# B&R Automation Studio project NAEUL004C00R13L518F00 (part 74)

#### InputRef.var - Do Not Change!!!
```iecst
(*2019-04-16*)
(**)
(*General*)
VAR
	p_udiRstErr : REFERENCE TO UDINT;
	p_bEn : REFERENCE TO BOOL;
	p_bDis : REFERENCE TO BOOL;
	p_bRun : REFERENCE TO BOOL;
	p_bStop : REFERENCE TO BOOL;
	p_bStep : REFERENCE TO BOOL;
END_VAR
(**)
(**)
VAR
	p_eUSCommMod1 : REFERENCE TO eMcSetCommMod;
	p_eUSCommMod2 : REFERENCE TO eMcSetCommMod;
	p_eUSCommMod3 : REFERENCE TO eMcSetCommMod;
	p_eDSCommMod1 : REFERENCE TO eMcSetCommMod;
	p_eDSCommMod2 : REFERENCE TO eMcSetCommMod;
	p_eDSCommMod3 : REFERENCE TO eMcSetCommMod;
END_VAR
(* *)
(**)
VAR
	p_tyBufferStat1 : REFERENCE TO tyBffrStat;
	p_tyBufferStat2 : REFERENCE TO tyBffrStat;
	p_tyBufferStat3 : REFERENCE TO tyBffrStat;
END_VAR
(**)
VAR
	p_dtBufferMagPresentTm1 : REFERENCE TO DATE_AND_TIME;
	p_dtBufferMagPresentTm2 : REFERENCE TO DATE_AND_TIME;
	p_dtBufferMagPresentTm3 : REFERENCE TO DATE_AND_TIME;
END_VAR
(* *)
VAR
	p_bUSHermesUSRdy1 : REFERENCE TO BOOL;
	p_bUSHermesUSGdRdy1 : REFERENCE TO BOOL;
	p_bUSHermesUSRdy2 : REFERENCE TO BOOL;
	p_bUSHermesUSGdRdy2 : REFERENCE TO BOOL;
	p_bUSHermesUSRdy3 : REFERENCE TO BOOL;
	p_bUSHermesUSGdRdy3 : REFERENCE TO BOOL;
	p_bUSSMEMAUSRdy1 : REFERENCE TO BOOL;
	p_bUSSMEMAUSRdy2 : REFERENCE TO BOOL;
	p_bUSSMEMAUSRdy3 : REFERENCE TO BOOL;
	p_bUSSMEMAGdBrdRdy1 : REFERENCE TO BOOL;
	p_bUSSMEMAGdBrdRdy2 : REFERENCE TO BOOL;
	p_bUSSMEMAGdBrdRdy3 : REFERENCE TO BOOL;
	p_bDSSMEMADSRdy1 : REFERENCE TO BOOL;
	p_bDSSMEMADSRdy2 : REFERENCE TO BOOL;
	p_bDSSMEMADSRdy3 : REFERENCE TO BOOL;
	p_bDSHermesDSRdy1 : REFERENCE TO BOOL;
	p_bDSHermesDSRdy2 : REFERENCE TO BOOL;
	p_bDSHermesDSRdy3 : REFERENCE TO BOOL;
	p_eULMod : REFERENCE TO eULMod;
	p_bBypsGdBadBrd : REFERENCE TO BOOL;
	p_bConvGdBrd : REFERENCE TO BOOL;
	p_usiLinkProdRcpCurrRcpMcMod : REFERENCE TO USINT;
	p_bOpsModGoneThrough : REFERENCE TO BOOL;
END_VAR
(**)
VAR
	p_tyParamTravLif : REFERENCE TO tyParamTravLifUL;
END_VAR
(**)
VAR
	p_sProgNm : REFERENCE TO STRING[15];
	p_bNtSettingsLoadDone : REFERENCE TO BOOL;
END_VAR
```

#### Local.var - Do Not Change!!!
```iecst
(*2019-04-16*)
(**)
(*Local Action, State & Status*)
VAR
	eStatus : eFBStatus := Idle;
	udiStatus : UDINT := 0;
END_VAR
(**)
(*Local Alarm*)
VAR
	tyAlmData : tyAlmDat;
	a_tyAlmText : ARRAY[10000..10099] OF tyAlmTxt;
END_VAR
(**)
(*Local Output*)
VAR
	sStepTxt : STRING[80];
	bPaused : BOOL;
END_VAR
(**)
(*Local Input*)
VAR
	udiRstErr : UDINT := 0;
	bEn : BOOL := TRUE;
	bDis : BOOL := FALSE;
	bRun : BOOL;
	bStop : BOOL;
	bStep : BOOL;
END_VAR
(*Insert your comment here.*)
VAR
	eUSCommMod1 : eMcSetCommMod;
	eUSCommMod2 : eMcSetCommMod;
	eUSCommMod3 : eMcSetCommMod;
	eDSCommMod1 : eMcSetCommMod;
	eDSCommMod2 : eMcSetCommMod;
	eDSCommMod3 : eMcSetCommMod;
	bUSSMEMAUSRdy3 : BOOL;
	bUSSMEMAGdBrdRdy3 : BOOL;
	udiUSPosAllwGo : UDINT := 99;
	udiDSPosAllwGo : UDINT := 99;
	a_bPosAllwSigOn : ARRAY[1..3] OF BOOL;
	a_udiPosAllwSum : ARRAY[1..3] OF UDINT;
	a_tyMagAllwBffrStat : ARRAY[1..3] OF tyBffrStat;
	a_udiMagAllwMagPresentTm : ARRAY[1..3] OF UDINT;
	a_udiMagAllwPriority : ARRAY[1..3] OF UDINT;
	udiMagPresentTm : UDINT;
	udiMagPresentTm1 : UDINT;
	bLocalUSRdy1 : BOOL;
	bLocalUSRdy2 : BOOL;
	bLocalUSRdy3 : BOOL;
	bLocalUSGdRdy1 : BOOL;
	bLocalUSGdRdy2 : BOOL;
	bLocalUSGdRdy3 : BOOL;
	bLocalDSRdy1 : BOOL;
	bLocalDSRdy2 : BOOL;
	bLocalDSRdy3 : BOOL;
	bDSHermesDSRdy1 : BOOL;
	bDSHermesDSRdy2 : BOOL;
	bDSHermesDSRdy3 : BOOL;
	bGdChk : BOOL;
	udi : UDINT;
END_VAR
(**)
(*Local*)
VAR
	sProgNm : STRING[80];
	bNtSettingsLoadDone : BOOL;
	bRstErr : BOOL;
	udiRstErrOld : UDINT;
	bInitDone : BOOL;
	bInitialDone : BOOL;
	eOpsStep : ePosUSAllwGoStep := ePosUSAllwGoStepNA;
	eGotoOpsStep : ePosUSAllwGoStep := ePosUSAllwGoUSCheck;
	eOpsStep1 : ePosDSAllwGoStep := ePosDSAllwGoStepNA;
	eGotoOpsStep1 : ePosDSAllwGoStep := ePosDSAllwGoDSCheck;
	fbMidChkDlyTm : TON := (PT:=T#1s);
	fbTopMidChkDlyTm : TON := (PT:=T#1s);
	udiCount : UDINT;
	udiCmpTm : UDINT;
	bBypsGdBadBrd : BOOL;
	eULMode : eULMod;
	bOpsModGonethrough : BOOL;
	udiModuleNum : UDINT;
END_VAR
```

### Simu.var - Change By Project
```iecst
(*2019-01-20*)
(**)
(*Action & State & Status*)
VAR
	p_SimuStat : UDINT;
	p_SimuStatus : UDINT;
	p_SimuStatTxt : UDINT;
END_VAR
(**)
(*Alarm*)
(**)
(*Output*)
VAR
	p_SimuSimuStatus : UDINT;
	p_SimuStatusRun : UDINT;
	p_SimuStatusStop : UDINT;
	p_SimuStatusCycleStop : UDINT;
	p_SimuStatusStep : UDINT;
	p_SimuRun : UDINT;
	p_SimuStop : UDINT;
	p_SimuStep : UDINT;
END_VAR
```

### Program Logical/Simulation/Simu (IEC, version 1.00.0) - 1.00.0 - 

#### Act_InitGlobal.st - Change By Project
```iecst
(** 2019-03-22 **)
ACTION Act_InitGlobal:

	(* Always Change If Project Change *)

	//Pass Data To Link
	p_eUISimuAct ACCESS p_UISimuAct;

	//Pass Data To Internal Use
	p_bLinkPaused ACCESS p_OpsPause;
	p_bNtSettingsLoadDone ACCESS p_StartupNtSettingsLoadDone;

	(* Always Change If Project Change *)

END_ACTION
```

#### InputRef_Link.var - Change By Project
```iecst
(*2019-01-20*)
(**)
VAR
	p_eUISimuAct : REFERENCE TO eSimulationsAction;
	p_bLinkPaused : REFERENCE TO BOOL;
END_VAR
```

#### Act_Link.st - Change By Project
```iecst
(** 2019-01-20 **)
ACTION Act_Link:

	p_bPaused := p_bLinkPaused;

END_ACTION
```

#### Local.var - Do Not Change!!!
```iecst
(*2019-04-30*)
(**)
(*Local Action, State & Status*)
VAR
	eAct : eSimulationsAction := SimulationsActIdle;
	eStat : eSimulationsAction := SimulationsActIdle;
	eStatus : eFBStatus := Idle;
	sStatTxt : STRING[200] := '';
	a_sStatText : ARRAY[0..50] OF STRING[200] := ['Idling','Starting Operations','Sequence Stopping Operations','Pause Operations In Step','Accepting New Data','Accepted New Data','Error Immediate Stop Operations',44('')];
END_VAR
(**)
(*Local Alarm*)
(**)
(*Local Output*)
VAR
	eSimuStatus : eSimulationsStatus := SimulationsStatusStop;
	bStatusRun : BOOL;
	bStatusStop : BOOL := TRUE;
	bStatusCycleStop : BOOL;
	bStatusStep : BOOL;
	bRun : BOOL;
	bStop : BOOL;
	bStep : BOOL;
END_VAR
(**)
(*Local Input*)
VAR
	udiRstErr : UDINT := 0;
	bPaused : BOOL;
	bNtSettingsLoadDone : BOOL := TRUE;
END_VAR
(**)
(*Local*)
VAR
	bRstErr : BOOL;
	udiRstErrOld : UDINT;
	bInitDone : BOOL;
	bInitialDone : BOOL;
	eStatOld : eSimulationsAction := SimulationsActIdle;
	usiStep : USINT;
END_VAR
```

### Simu1.var - Change By Project
```iecst
(*2022-10-17*)
(**)
(*Action & State & Status*)
(**)
(*Alarm*)
(**)
(*Output*)
VAR
	p_Simu1Paused : UDINT;
END_VAR
(**)
VAR
	p_Simu1InShutterAct : UDINT;
	p_Simu1OutShutterAct : UDINT;
	p_Simu1OutShutterAct2 : UDINT;
	p_Simu1OutShutterAct3 : UDINT;
END_VAR
```

### Simu1.typ - Do Not Change!!!
```iecst
(*2018-12-11*)
(**)
(*Sequence*)

TYPE
	eSimuRunStep :
		(
		SimuStepNA,
		SimuStepChkPshrRetSen,
		SimuStepChkSen,
		SimuStepInShutterRet,
		SimuStepInShutterExt,
		SimuStepOutShutterRet,
		SimuStepOutShutterExt
		);
END_TYPE
```

### Program Logical/Simulation/Simu1 (IEC) - 1.00.0 - 

#### InputRef.var
```iecst
(*2022-10-17*)
(**)
(*General*)
VAR
	p_udiRstErr : REFERENCE TO UDINT;
	p_bEn : REFERENCE TO BOOL;
	p_bDis : REFERENCE TO BOOL;
	p_bRun : REFERENCE TO BOOL;
	p_bStop : REFERENCE TO BOOL;
	p_bStep : REFERENCE TO BOOL;
END_VAR
(**)
(**)
VAR
	p_eInShuttStat : REFERENCE TO ePneuAction;
	p_eInShuttStatus : REFERENCE TO eFBStatus;
	p_eOutShuttStat : REFERENCE TO ePneuAction;
	p_eOutShuttStatus : REFERENCE TO eFBStatus;
	p_eOutShutt2Stat : REFERENCE TO ePneuAction;
	p_eOutShutt2Status : REFERENCE TO eFBStatus;
	p_eOutShutt3Stat : REFERENCE TO ePneuAction;
	p_eOutShutt3Status : REFERENCE TO eFBStatus;
END_VAR
(**)
(**)
VAR
	p_sProgNm : REFERENCE TO STRING[15];
	p_bNtSettingsLoadDone : REFERENCE TO BOOL;
END_VAR
```

#### Local.var
```iecst
(*2022-10-17*)
(**)
(*Local Action, State & Status*)
VAR
	eStatus : eFBStatus := Idle;
	udiStatus : UDINT := 0;
END_VAR
(**)
(*Local Alarm*)
VAR
	tyAlmData : tyAlmDat;
	a_tyAlmText : ARRAY[10000..10099] OF tyAlmTxt;
END_VAR
(**)
(*Local Output*)
VAR
	sStepTxt : STRING[80];
	bPaused : BOOL;
	ePshrAct : eMtrPshrAction;
	eInShutterAct : ePneuAction;
	eOutShutterAct : ePneuAction;
	eOutShutterAct2 : ePneuAction;
	eOutShutterAct3 : ePneuAction;
END_VAR
(**)
(*Local Input*)
VAR
	udiRstErr : UDINT := 0;
	bEn : BOOL := TRUE;
	bDis : BOOL := FALSE;
	bRun : BOOL;
	bStop : BOOL;
	bStep : BOOL;
END_VAR
(**)
(**)
VAR
	eInShutt1Stat : ePneuAction;
	eInShutt1Status : eFBStatus;
	eOutShutt2Stat : ePneuAction;
	eOutShutt2Status : eFBStatus;
	eOutShuttStat : ePneuAction;
	eOutShuttStatus : eFBStatus;
	eOutShutt3Stat : ePneuAction;
	eOutShutt3Status : eFBStatus;
END_VAR
(**)
VAR
	sProgNm : STRING[15];
	bNtSettingsLoadDone : BOOL := TRUE;
END_VAR
(**)
(*Local*)
VAR
	bRstErr : BOOL;
	udiRstErrOld : UDINT;
	bInitDone : BOOL;
	bInitialDone : BOOL;
	eSimuStep : eSimuRunStep := SimuStepNA;
	eSimuGotoStep : eSimuRunStep := SimuStepChkSen;
	fbShutterExtDlyTm : TON := (PT:=T#200ms);
	udiModuleNum : UDINT;
END_VAR
```

#### Act_InitGlobal.st
```iecst
(** 2022-10-17 **)
ACTION Act_InitGlobal:

	(* Always Change If Project Change *)

	//Pass Data To Link

	//Pass Data To Internal Use
	p_udiRstErr ACCESS p_RstErrReset;
	p_bRun ACCESS p_SimuRun;
	p_bStop ACCESS p_SimuStop;
	p_bStep ACCESS p_SimuStep;
	p_bNtSettingsLoadDone ACCESS p_StartupNtSettingsLoadDone;

	p_eInShuttStat ACCESS p_Pneu2SenInShutterStat;
	p_eInShuttStatus ACCESS p_Pneu2SenInShutterStatus;

	p_eOutShuttStat ACCESS p_Pneu2SenOutShutterStat;
	p_eOutShuttStatus ACCESS p_Pneu2SenOutShutterStatus;

	p_eOutShutt2Stat ACCESS p_Pneu2SenOutShutterStat2;
	p_eOutShutt2Status ACCESS p_Pneu2SenOutShutterStatus2;

	p_eOutShutt3Stat ACCESS p_Pneu2SenOutShutterStat3;
	p_eOutShutt3Status ACCESS p_Pneu2SenOutShutterStatus3;

	//p_sProgNm ACCESS p_NtParamSimuTeleNOProgNm;

	(* Always Change If Project Change *)

END_ACTION
```

#### Act_Initial.st
```iecst
(** 2022-10-17 **)
ACTION Act_Initial:

	//Initial

END_ACTION
```

#### Act_InitLocal.st
```iecst
(** 2022-10-17 **)
ACTION Act_InitLocal:

	//Input Reference Link To Local Variable
	p_udiRstErr ACCESS ADR(udiRstErr);
	p_bEn ACCESS ADR(bEn);
	p_bDis ACCESS ADR(bDis);
	p_bRun ACCESS ADR(bRun);
	p_bStop ACCESS ADR(bStop);
	p_bStep ACCESS ADR(bStep);

	p_eInShuttStat ACCESS ADR(eInShutt1Stat);
	p_eInShuttStatus ACCESS ADR(eInShutt1Status);
	p_eOutShuttStat ACCESS ADR(eOutShuttStat);
	p_eOutShuttStatus ACCESS ADR(eOutShuttStatus);
	p_eOutShutt2Stat ACCESS ADR(eOutShutt2Stat);
	p_eOutShutt2Status ACCESS ADR(eOutShutt2Status);
	p_eOutShutt3Stat ACCESS ADR(eOutShutt3Stat);
	p_eOutShutt3Status ACCESS ADR(eOutShutt3Status);

	p_sProgNm ACCESS ADR(sProgNm);
	p_bNtSettingsLoadDone ACCESS ADR(bNtSettingsLoadDone);

END_ACTION
```

#### Act_Link.st
```iecst
(** 2022-10-17 **)
ACTION Act_Link:

END_ACTION
```

#### Act_LinkEn.st
```iecst
(** 2022-10-17 **)
ACTION Act_LinkEn:

	//Link bPrep, bEn & bDis

END_ACTION
```

#### Cyclic.st
```iecst
(** 2022-10-17 **)
PROGRAM _CYCLIC

	IF bInitDone = FALSE THEN
		bInitDone	:= TRUE;

		Act_InitLocal;
		Act_InitGlobal;

	ELSIF bInitialDone = FALSE THEN
		IF p_bNtSettingsLoadDone = TRUE THEN
			bInitialDone	:= TRUE;

			Act_Initial;
		END_IF

	ELSE

		Act_RstErr;
		Act_LinkEn;
		Act_Link;
		Act_Background;
		Act_Alarm;

	END_IF

END_PROGRAM
```

#### Init.st
```iecst
(** 2022-10-17 **)
PROGRAM _INIT

	(* Always Change If Project Change *)

	//Pass Address To Global Address For External Use
	//Action, State & Status

	//Alarm

	//Output
	p_Simu1Paused					:= ADR(bPaused);

	p_Simu1InShutterAct				:= ADR(eInShutterAct);
	p_Simu1OutShutterAct			:= ADR(eOutShutterAct);
	p_Simu1OutShutterAct2			:= ADR(eOutShutterAct2);
	p_Simu1OutShutterAct3			:= ADR(eOutShutterAct2);

	(* Always Change If Project Change *)

END_PROGRAM
```

#### Program Logical/Simulation/Simu1/Sequence

##### Act_OpsInitial.st
```iecst
(** 2019-01-16 **)
ACTION Act_OpsInitial:

	eSimuGotoStep	:= SimuStepChkSen;
	eSimuStep		:= SimuStepNA;

END_ACTION
```

##### Act_OpsRst.st
```iecst
(** 2022-10-17 **)
ACTION Act_OpsRst:

	eOutShutterAct			:= PneuActIdle;
	eOutShutterAct2			:= PneuActIdle;
	eOutShutterAct3			:= PneuActIdle;
	fbShutterExtDlyTm(IN:=FALSE);

END_ACTION
```

##### Act_OpsRun.st
```iecst
(** 2022-10-17 **)
ACTION Act_OpsRun:

	IF eSimuGotoStep <> eSimuStep THEN

		CASE eSimuGotoStep OF

			ELSE
				eSimuStep	:= eSimuGotoStep;

		END_CASE

	END_IF

	IF eSimuGotoStep = eSimuStep THEN

		IF bPaused = FALSE THEN

			CASE eSimuStep OF

			SimuStepOutShutterExt:

						eOutShutterAct	:= PneuActExt;
						eOutShutterAct2 := PneuActExt;
						eOutShutterAct3	:= PneuActExt;

					IF 	p_eOutShuttStat = PneuActExt AND p_eOutShuttStatus = Done AND
						p_eOutShutt2Stat = PneuActExt AND p_eOutShutt2Status = Done AND
						p_eOutShutt3Stat = PneuActExt AND p_eOutShutt3Status = Done THEN

						eOutShutterAct	:= PneuActIdle;
						eOutShutterAct2 := PneuActIdle;
						eOutShutterAct3 := PneuActIdle;

						fbShutterExtDlyTm(IN:=TRUE);
						IF fbShutterExtDlyTm.Q THEN
							fbShutterExtDlyTm(IN:=FALSE);
						eSimuGotoStep	:= SimuStepOutShutterRet;
						END_IF
						bPaused				:= p_bStop OR p_bStep;
					END_IF

				SimuStepOutShutterRet:

					eOutShutterAct	:= PneuActRet;
					eOutShutterAct2 := PneuActRet;
					eOutShutterAct3 := PneuActRet;
					IF 	p_eOutShuttStat = PneuActRet AND p_eOutShuttStatus = Done AND
						p_eOutShutt2Stat = PneuActRet AND p_eOutShutt2Status = Done AND
						p_eOutShutt3Stat = PneuActRet AND p_eOutShutt3Status = Done	 THEN

						eOutShutterAct	:= PneuActIdle;
						eOutShutterAct2 := PneuActIdle;
						eOutShutterAct3 := PneuActIdle;

						fbShutterExtDlyTm(IN:=TRUE);
						IF fbShutterExtDlyTm.Q THEN
							fbShutterExtDlyTm(IN:=FALSE);
						eSimuGotoStep	:= SimuStepOutShutterExt;
						END_IF
						bPaused			:= p_bStop OR p_bStep;
					END_IF

			END_CASE

		END_IF
	END_IF

END_ACTION
```

### Simu2.var - Change By Project
```iecst
(*2022-10-17*)
(**)
(*Action & State & Status*)
(**)
(*Alarm*)
(**)
(*Output*)
VAR
	p_Simu2Paused : UDINT;
END_VAR
(**)
VAR
	p_Simu2DispCyclTmBffr1 : UDINT;
	p_Simu2DispCyclTmBffr2 : UDINT;
	p_Simu2DispCyclTmBffr3 : UDINT;
END_VAR
```

### Simu2.typ - Do Not Change!!!
```iecst
(*2018-12-11*)
(**)
(*Sequence*)
(*Display Buffer*)

TYPE
	tyDispBffrCycTm : 	STRUCT  (*Buffer Display in HMI*)
		diDispIdxSt : DINT; (*Start Index Display in HMI*)
		diDispIdxEnd : DINT; (*End Index Display in HMI*)
		a_tyDispBffrDat : ARRAY[1..c_diDispBffrSize]OF tyDispBffrCycTmDat; (*Array of Buffer Data Display in HMI*)
	END_STRUCT;
	tyDispBffrCycTmDat : 	STRUCT  (*Display Buffer Data*)
		sSlttoSltIdx : STRING[80]; (*Slot Index*)
		sCycleTm : STRING[80]; (*Board Loaded Time*)
		dwColor : DWORD; (*Color For Good & Bad Board*)
	END_STRUCT;
END_TYPE
```

### Program Logical/Simulation/Simu2 (IEC) - 1.00.0 - 

#### InputRef.var
```iecst
(*2022-10-17*)
(**)
(*General*)
VAR
	p_udiRstErr : REFERENCE TO UDINT;
	p_bEn : REFERENCE TO BOOL;
	p_bDis : REFERENCE TO BOOL;
	p_bRun : REFERENCE TO BOOL;
	p_bStop : REFERENCE TO BOOL;
	p_bStep : REFERENCE TO BOOL;
END_VAR
(**)
VAR
	p_diSltCap : REFERENCE TO DINT;
	p_diBffrTtlSlt : REFERENCE TO DINT;
	p_bTravDPosDiff : REFERENCE TO BOOL;
	p_bTravEPosDiff : REFERENCE TO BOOL;
	p_bTravFPosDiff : REFERENCE TO BOOL;
	p_bLifterBtmSltAPosDiff : REFERENCE TO BOOL;
	p_bLifterBtmSltBPosDiff : REFERENCE TO BOOL;
	p_bLifterBtmSltCPosDiff : REFERENCE TO BOOL;
	p_diLifterBtmCurrSltA : REFERENCE TO DINT;
	p_diLifterBtmCurrSltB : REFERENCE TO DINT;
	p_diLifterBtmCurrSltC : REFERENCE TO DINT;
	p_eOpsTravLifOpsStep : REFERENCE TO eTravLifULStep;
	p_eOpsTravLifGotoOpsStep : REFERENCE TO eTravLifULStep;
	p_dtTimeCurrDT : REFERENCE TO DATE_AND_TIME;
	p_uiTimeCurrDTStructMS : REFERENCE TO UINT;
	p_tyDispCycTmBffr : REFERENCE TO tyDispBffrCycTm;
	p_tyBuffer : REFERENCE TO tyBffr;
	p_diSlotCount : REFERENCE TO DINT;
END_VAR
(**)
(**)
(**)
VAR
	p_sProgNm : REFERENCE TO STRING[15];
	p_bNtSettingsLoadDone : REFERENCE TO BOOL;
END_VAR
```

#### Local.var
```iecst
(*2022-10-17*)
(**)
(*Local Action, State & Status*)
VAR
	eStatus : eFBStatus := Idle;
	udiStatus : UDINT := 0;
END_VAR
(**)
(*Local Alarm*)
VAR
	tyAlmData : tyAlmDat;
	a_tyAlmText : ARRAY[10000..10099] OF tyAlmTxt;
END_VAR
(**)
(*Local Output*)
VAR
	sStepTxt : STRING[80];
	bPaused : BOOL;
END_VAR
(**)
(*Local Input*)
VAR
	udiRstErr : UDINT := 0;
	bEn : BOOL := TRUE;
	bDis : BOOL := FALSE;
	bRun : BOOL;
	bStop : BOOL;
	bStep : BOOL;
END_VAR
(**)
VAR
	diSltCap : DINT := 1;
	diBffrTtlSlt : DINT;
	tyDispCycTmBffr : tyDispBffrCycTm;
	sCurrSlotTransition : STRING[80];
	diCnt : DINT;
	diSlotCount : DINT;
	diDispIdx : DINT;
	dicntr1 : DINT;
	a_tyDispCycTmBffr : ARRAY[0..2] OF tyDispBffrCycTm;
	tyBuffer : tyBffr;
	dtCycleTim : TIME;
	dtDumyTim : TIME := T#0ms;
	dwGdColor : DWORD;
	dwNAColor : DWORD;
	tAccumulateTimer : TIME;
	tPrevTim : TIME;
	sSltnumber : STRING[80];
	TtestPrevTim : DATE_AND_TIME;
	tTesttime : TIME;
	teststep : USINT;
	testpos : USINT;
END_VAR
(**)
(**)
VAR
	sProgNm : STRING[15];
	bNtSettingsLoadDone : BOOL := TRUE;
END_VAR
(**)
(*Local*)
VAR
	bRstErr : BOOL;
	udiRstErrOld : UDINT;
	bInitDone : BOOL;
	bInitialDone : BOOL;
	udiModuleNum : UDINT;
END_VAR
```

#### Act_Alarm.st
```iecst
(** 2022-10-17 **)
ACTION Act_Alarm:

	//Error
	IF EDGEPOS(eStatus = Error) THEN

		tyAlmData.sProgNm		:= p_sProgNm;
		tyAlmData.udiCode		:= udiStatus;
		tyAlmData.eSeverity		:= AlmSeverityError;
		tyAlmData.udiRunTime	:= tyAlmData.udiRunTime + 1;
		tyAlmData.bAlm			:= TRUE;
		tyAlmData.udiModuleNum  := udiModuleNum;
		g_sSimu1ProgNm		:= p_sProgNm;
		//Get Error Message
		IF tyAlmData.udiCode < 10000 OR tyAlmData.udiCode > 10099 THEN
			tyAlmData.sAlmMsg	:= 'Unknown';
			tyAlmData.sRcyMsg	:= 'Unknown';
		ELSE
			tyAlmData.sAlmMsg	:= a_tyAlmText[tyAlmData.udiCode].sAlmText;
			tyAlmData.sRcyMsg	:= a_tyAlmText[tyAlmData.udiCode].sRcyText;
		END_IF

	ELSIF bRstErr AND (tyAlmData.udiCode <> 0) THEN

		tyAlmData.udiCode		:= 0;
		tyAlmData.eSeverity		:= AlmSeverityNA;
		tyAlmData.sAlmMsg		:= '';
		tyAlmData.sRcyMsg		:= '';
		tyAlmData.bAlm			:= FALSE;
	END_IF

END_ACTION
```

#### Act_Background.st
```iecst
(** 2022-10-17 **)
ACTION Act_Background:

	//Reset bPaused
	IF EDGENEG(p_bStop OR p_bStep) THEN
		bPaused	:= FALSE;
	END_IF

	IF eStatus <> Error AND p_bRun = TRUE THEN
		IF (p_bEn = TRUE) AND (p_bDis = FALSE) THEN
			Act_OpsRun;
		ELSE
			bPaused	:= p_bStop OR p_bStep;
		END_IF

		IF EDGEPOS(p_bEn = FALSE OR p_bDis = TRUE) THEN
			Act_OpsRst;
		END_IF

	ELSIF eStatus <> Error THEN
		sStepTxt	:= 'Stop';
	ELSE
		sStepTxt	:= 'Error';
	END_IF

	//Reset
	IF EDGENEG(p_bRun) OR EDGEPOS(eStatus = Error) THEN
		Act_OpsInitial;
		Act_OpsRst;
	END_IF

	//Reset Error
	IF (eStatus = Error) AND bRstErr THEN
		eStatus		:= Idle;
		udiStatus	:= 0;
	END_IF

END_ACTION
```

#### Act_InitGlobal.st
```iecst
(** 2022-10-17 **)
ACTION Act_InitGlobal:

	(* Always Change If Project Change *)

	//Pass Data To Link

	//Pass Data To Internal Use
	p_udiRstErr ACCESS p_RstErrReset;
	p_bRun ACCESS p_SimuRun;
	p_bStop ACCESS p_SimuStop;
	p_bStep ACCESS p_SimuStep;
	p_bNtSettingsLoadDone ACCESS p_StartupNtSettingsLoadDone;

	//OpsCycleTim
	p_bTravDPosDiff ACCESS p_TravDPosDiff;
	p_bTravEPosDiff ACCESS p_TravEPosDiff;
	p_bTravFPosDiff ACCESS p_TravFPosDiff;
	p_bLifterBtmSltAPosDiff ACCESS p_LifterBtmSltAPosDiff;
	p_bLifterBtmSltBPosDiff ACCESS p_LifterBtmSltBPosDiff;
	p_bLifterBtmSltCPosDiff ACCESS p_LifterBtmSltCPosDiff;
	p_diLifterBtmCurrSltA ACCESS p_LifterBtmCurrSltA;
	p_diLifterBtmCurrSltB ACCESS p_LifterBtmCurrSltB;
	p_diLifterBtmCurrSltC ACCESS p_LifterBtmCurrSltC;

	p_eOpsTravLifOpsStep ACCESS p_OpsTravLifOpsStep;
	p_eOpsTravLifGotoOpsStep ACCESS p_OpsTravLifGotoOpsStep;
	p_dtTimeCurrDT ACCESS p_TimeCurrDT	;
	p_diBffrTtlSlt ACCESS p_MagRcpCurrRcpTtlSlt;
    p_uiTimeCurrDTStructMS ACCESS p_TimeCurrDTStructMS;
	//p_sProgNm ACCESS p_NtParamSimuTeleNOProgNm;

	(* Always Change If Project Change *)

END_ACTION
```

#### Act_InitLocal.st
```iecst
(** 2022-10-17 **)
ACTION Act_InitLocal:

	//Input Reference Link To Local Variable
	p_udiRstErr ACCESS ADR(udiRstErr);
	p_bEn ACCESS ADR(bEn);
	p_bDis ACCESS ADR(bDis);
	p_bRun ACCESS ADR(bRun);
	p_bStop ACCESS ADR(bStop);
	p_bStep ACCESS ADR(bStep);

	p_diSltCap ACCESS ADR(diSltCap);
	p_diBffrTtlSlt ACCESS ADR(diBffrTtlSlt);
	p_tyDispCycTmBffr ACCESS ADR(tyDispCycTmBffr);
	p_tyBuffer ACCESS ADR(tyBuffer);
	p_diSltCap ACCESS ADR(diSltCap);
	p_diSlotCount ACCESS ADR(diCnt);

	p_sProgNm ACCESS ADR(sProgNm);
	p_bNtSettingsLoadDone ACCESS ADR(bNtSettingsLoadDone);

END_ACTION
```

#### Act_Link.st
```iecst
(** 2022-10-17 **)
ACTION Act_Link:

 	//tTesttime := UINT_TO_TIME(p_uiTimeCurrDTStructMS);
END_ACTION
```

#### Act_RstErr.st
```iecst
(** 2022-10-17 **)
ACTION Act_RstErr:

	IF p_udiRstErr <> udiRstErrOld THEN
		bRstErr			:= TRUE;
		udiRstErrOld	:= p_udiRstErr;
	ELSE
		bRstErr			:= FALSE;
	END_IF

END_ACTION
```

#### Init.st
```iecst
(** 2022-10-17 **)
PROGRAM _INIT

	(* Always Change If Project Change *)

	//Pass Address To Global Address For External Use
	//Action, State & Status

	//Alarm

	//Output
	p_Simu2Paused					:= ADR(bPaused);

	p_Simu2DispCyclTmBffr1					:= ADR(a_tyDispCycTmBffr[0]);
	p_Simu2DispCyclTmBffr2					:= ADR(a_tyDispCycTmBffr[1]);
	p_Simu2DispCyclTmBffr3					:= ADR(a_tyDispCycTmBffr[2]);

	(* Always Change If Project Change *)

END_PROGRAM
```

#### Act_OpsInitial.st - Do Not Change!!!
```iecst
(** 2019-01-16 **)
ACTION Act_OpsInitial:

END_ACTION
```

#### Act_OpsRun.st
```iecst
(** 2022-10-17 **)
ACTION Act_OpsRun:

	//A15<-A13 | timetaken

	IF (p_eOpsTravLifOpsStep =  TravLifULStepExitBrd AND p_eOpsTravLifGotoOpsStep = TravLifULStepOutletPneuCls)  THEN
		memset(ADR(dtCycleTim),0,SIZEOF(dtCycleTim));
		IF FIND(sCurrSlotTransition,'<-') <> 0 THEN
			sCurrSlotTransition := LEFT( sCurrSlotTransition , FIND(sCurrSlotTransition,'<-') - 1);
		END_IF

		IF NOT(p_bTravDPosDiff  OR p_bLifterBtmSltAPosDiff)   THEN
			itoa(DINT_TO_INT(p_diLifterBtmCurrSltA),ADR(sSltnumber));
			sCurrSlotTransition := CONCAT(CONCAT(CONCAT('A',sSltnumber),'<-'),sCurrSlotTransition);
			dtCycleTim := ((DT_TO_TIME(p_dtTimeCurrDT) +UINT_TO_TIME(p_uiTimeCurrDTStructMS) -tPrevTim )+ tAccumulateTimer);
			tPrevTim 			:= DT_TO_TIME(p_dtTimeCurrDT) + UINT_TO_TIME(p_uiTimeCurrDTStructMS);
		ELSIF NOT(p_bTravEPosDiff OR p_bLifterBtmSltBPosDiff )  THEN
			itoa(DINT_TO_INT(p_diLifterBtmCurrSltB),ADR(sSltnumber));
			sCurrSlotTransition := CONCAT(CONCAT(CONCAT('B',sSltnumber),'<-'),sCurrSlotTransition);
			dtCycleTim := ((DT_TO_TIME(p_dtTimeCurrDT) +UINT_TO_TIME(p_uiTimeCurrDTStructMS) -tPrevTim )+ tAccumulateTimer);
			tPrevTim 			:= DT_TO_TIME(p_dtTimeCurrDT) + UINT_TO_TIME(p_uiTimeCurrDTStructMS);
		ELSIF NOT(p_bTravFPosDiff OR p_bLifterBtmSltCPosDiff)  THEN
			itoa(DINT_TO_INT(p_diLifterBtmCurrSltC),ADR(sSltnumber));
			sCurrSlotTransition := CONCAT(CONCAT(CONCAT('C',sSltnumber),'<-'),sCurrSlotTransition);
			dtCycleTim := ((DT_TO_TIME(p_dtTimeCurrDT) +UINT_TO_TIME(p_uiTimeCurrDTStructMS) -tPrevTim )+ tAccumulateTimer); //+ tAccumulateTimer
			tPrevTim 			:= DT_TO_TIME(p_dtTimeCurrDT) + UINT_TO_TIME(p_uiTimeCurrDTStructMS);
		ELSE
			sCurrSlotTransition := '';
			tPrevTim 			:= 0;
		END_IF
		IF memcmp(ADR(dtCycleTim),ADR(dtDumyTim),SIZEOF(dtCycleTim)) <> 0 THEN ;
			Act_DispBffr;
		END_IF
	ELSIF (p_eOpsTravLifGotoOpsStep = TravLifULStepUSComm AND (p_eOpsTravLifOpsStep = TravLifULStepInletPneuOpn OR p_eOpsTravLifOpsStep= TravLifULStepTravLifMov ))  THEN
			IF tPrevTim <> 0 THEN
				tAccumulateTimer := (DT_TO_TIME(p_dtTimeCurrDT)+UINT_TO_TIME(p_uiTimeCurrDTStructMS) ) - tPrevTim  ;
			END_IF
	ELSIF (p_eOpsTravLifOpsStep =  TravLifULStepUSComm AND p_eOpsTravLifGotoOpsStep = TravLifULStepEntBrd) THEN
			tPrevTim		  := DT_TO_TIME(p_dtTimeCurrDT) +UINT_TO_TIME(p_uiTimeCurrDTStructMS) ;
	END_IF

END_ACTION
```

#### Act_OpsRst.st - Do Not Change!!!
```iecst
(** 2022-10-17 **)
ACTION Act_OpsRst:

	tPrevTim := 0;
	tAccumulateTimer := 0;

END_ACTION
```

#### Act_DispBffr.st
```iecst
(** 2022-10-17 **)
ACTION Act_DispBffr:

	memset(ADR(p_tyDispCycTmBffr) , 0 , SIZEOF(p_tyDispCycTmBffr));
	IF NOT(p_bTravDPosDiff  OR p_bLifterBtmSltAPosDiff) THEN
		p_tyDispCycTmBffr ACCESS ADR(a_tyDispCycTmBffr[0]);
		p_tyBuffer ACCESS p_Buffer1Bffr;
		p_diSlotCount ACCESS p_LifterBtmCurrSltA;
	ELSIF NOT(p_bTravEPosDiff OR p_bLifterBtmSltBPosDiff ) THEN
		p_tyDispCycTmBffr ACCESS ADR(a_tyDispCycTmBffr[1]);
		p_tyBuffer ACCESS p_Buffer2Bffr;
		p_diSlotCount ACCESS p_LifterBtmCurrSltB;
	ELSIF NOT(p_bTravFPosDiff OR p_bLifterBtmSltCPosDiff) THEN
		p_tyDispCycTmBffr ACCESS ADR(a_tyDispCycTmBffr[2]);
		p_tyBuffer ACCESS p_Buffer3Bffr;
		p_diSlotCount ACCESS p_LifterBtmCurrSltC;
	END_IF
	diCnt	:= 0;
	dwNAColor := 0;
	dwGdColor := 1;

	FOR dicntr1 := 1 TO p_diBffrTtlSlt DO

		//Get Display Index
		diDispIdx	:= p_diBffrTtlSlt * p_diSltCap - diCnt; //p_diLifterBtmCurrSltA
		diCnt := diCnt +1;

		IF p_diSlotCount = diCnt AND p_tyBuffer.a_tyBffrDat[diCnt].bSltForBrd AND p_tyBuffer.a_tyBffrDat[diCnt].bBrdAvl AND p_tyBuffer.a_tyBffrDat[diCnt].a_tySubBffrDat[1].bSubForBrd AND p_tyBuffer.a_tyBffrDat[diCnt].a_tySubBffrDat[1].bBrdAvl THEN
			ascTIME(dtCycleTim , ADR(p_tyDispCycTmBffr.a_tyDispBffrDat[diDispIdx].sCycleTm) , SIZEOF(p_tyDispCycTmBffr.a_tyDispBffrDat[diDispIdx].sCycleTm));
			p_tyDispCycTmBffr.a_tyDispBffrDat[diDispIdx].dwColor	:= dwGdColor;
			p_tyDispCycTmBffr.a_tyDispBffrDat[diDispIdx].sSlttoSltIdx := sCurrSlotTransition;
		ELSE
			p_tyDispCycTmBffr.a_tyDispBffrDat[diDispIdx].dwColor	:= dwNAColor;
			p_tyDispCycTmBffr.a_tyDispBffrDat[diDispIdx].sSlttoSltIdx := DINT_TO_STRING(dicntr1);
		END_IF

	END_FOR

	p_tyDispCycTmBffr.diDispIdxSt	:= 1;
	p_tyDispCycTmBffr.diDispIdxEnd	:= p_diBffrTtlSlt * p_diSltCap;

END_ACTION
```

### OpCon.typ - Do Not Change!!!
```iecst
(*2019-05-04*)
(**)
(*Action*)

TYPE
	eOpConAction :
		(
		OpConActIdle,
		OpConActBGStartRun,
		OpConActBGStopRun,
		OpConActDeleteOldLog,
		OpConActCreateDir,
		OpConActWriteRetain,
		OpConActReadRetain,
		OpConActWriteConfig,
		OpConActReadConfig
		);
END_TYPE
```

### OpCon.var - Change By Project
```iecst
(*2019-06-10*)
(**)
(*Action & State & Status*)
VAR
	p_OpConStat : UDINT;
	p_OpConStatus : UDINT;
	p_OpConStatTxt : UDINT;
END_VAR
(**)
(*Alarm*)
VAR
	p_OpConAlmData : UDINT;
	p_OpConAlmData1 : UDINT;
	p_OpConInfoData : UDINT;
END_VAR
(**)
(*Output*)
VAR
	p_OpConTableDataBrdAvl : UDINT;
	p_OpConTableDataBrdAvlTtlIdx : UDINT;
	p_OpConConnected : UDINT;
	p_OpConHandshakeDone : UDINT;
	p_OpConOverWriteSlt : UDINT;
	p_OpConOverWriteWidth : UDINT;
	p_OpConReqRecipeNm : UDINT;
	p_OpConReqWidthInUM : UDINT;
	p_OpConInternalSnd : UDINT;
	p_OpConPartRcvRetCode : UDINT;
	p_OpConPlcGrabRcvCode : UDINT;
END_VAR
```

### Program Logical/OpCon/OpCon (IEC, version 1.00.0) - 1.00.0 - NtHermes v5.00.0 , NtTCP v5.00.0 , NtMessage v5.00.0

#### Init.st - Change By Project
```iecst
(** 2019-06-10 **)
PROGRAM _INIT

	(* Always Change If Project Change *)

	//Pass Address To Global Address For External Use
	//Action, State & Status
	p_OpConStat		:= ADR(eStat);
	p_OpConStatus	:= ADR(eMainStatus);
	p_OpConStatTxt	:= ADR(sStatTxt);

	//Alarm
	p_OpConAlmData	:= ADR(tyAlmData);
	p_OpConAlmData1	:= ADR(tyAlmData1);
	p_OpConInfoData	:= ADR(tyInfoData);

	//Output
	p_OpConTableDataBrdAvl			:= ADR(a_tyXMLTableDataBrdAvl);
	p_OpConTableDataBrdAvlTtlIdx	:= ADR(iXMLTableDataBrdAvlTtlIdx);
	p_OpConConnected				:= ADR(bConnected);
	p_OpConHandshakeDone			:= ADR(bHandshakeDone);
	p_OpConOverWriteSlt			:= ADR(bOverWriteSlt);
	p_OpConOverWriteWidth		:= ADR(bOverWriteWidth);
	p_OpConReqRecipeNm			:= ADR(sReqRecipeNm);
	p_OpConReqWidthInUM			:= ADR(diReqWidthInUM);
	p_OpConInternalSnd			:= ADR(sInternalSnd);

	p_OpConPartRcvRetCode		:= ADR(tyPartReceive);
	p_OpConPlcGrabRcvCode			:= ADR(tyPlcGrab);
	(* Always Change If Project Change *)

END_PROGRAM
```

#### Act_InitGlobal.st - Change By Project
```iecst
(** 2019-06-28 **)
ACTION Act_InitGlobal:

	(* Always Change If Project Change *)

	//Pass Data To Link
	p_bLinkStartupRun ACCESS p_StartupRun;

	p_eLinkConvDir ACCESS p_NtParamProjConvDir;
	p_bLinkDILeftSen ACCESS p_DIConvLftSen;
	p_bLinkDIRightSen ACCESS p_DIConvRgtSen;
	p_tyLinkAlarmCurrList ACCESS p_AlarmCurrList;
	p_bLinkOpConEn ACCESS p_McParamOpConEn;

	//Pass Data To Internal Use
	p_udiRstErr ACCESS p_RstErrReset;
	p_bPrep ACCESS p_NtParamProjOpConPrep;
//	p_bEn ACCESS p_McParamOpConEn;
	p_sIPAddr ACCESS p_HWInfoIPAddr; //client
	p_sSvrIPAddr ACCESS p_McParamOpConIP;
	p_uiSvrIPPort ACCESS p_McParamOpConPort;
	p_tyDTStructure ACCESS p_TimeCurrDTStruct;
	p_dtCurrDT ACCESS p_TimeCurrDT;

	p_sRecipeNm ACCESS p_ProdRcpCurrRcp0Nm;
	p_diWidthInUM ACCESS p_ProdRcpCurrRcp0Width;
	p_bOpsRun ACCESS p_OpsRun;
	p_bNtSettingsLoadDone ACCESS p_StartupNtSettingsLoadDone;
	pa_tyProdRcpList ACCESS p_ProdRcpCurrList;
	p_tyProdRcpCurrRcp ACCESS p_ProdRcpCurrRcp0;

	p_tyOpConLocation ACCESS p_McParamOpConParam;
	p_bOpsTravLifULExitBrd ACCESS p_OpsTravLifULExitBrd;
	p_tyOpsTravLifULMsgReq ACCESS p_OpsTravLifULMsgReq;
	p_sOpsTravLifULBarcode ACCESS p_OpsTravLifULBarcode;
	p_tyOpsTravLifULPartProcessItms ACCESS p_OpsTravLifULPartProcessItms; //new
	pas_OpsTravLifULMagEntered ACCESS p_OpsTravLifULMagEntered;
	p_tyOpsMagConvUL1MsgReq ACCESS p_OpsMagConvUL1MsgReq;
	(* Always Change If Project Change *)

END_ACTION
```

#### InputRef_Link.var - Change By Project
```iecst
(*2019-04-16*)
(**)
VAR
	p_bLinkStartupRun : REFERENCE TO BOOL;
	bOpConRun : BOOL;
	bOpConStop : BOOL;
END_VAR
(**)
VAR
	p_eLinkConvDir : REFERENCE TO eConvDir;
	p_bLinkDILeftSen : REFERENCE TO BOOL;
	p_bLinkDIRightSen : REFERENCE TO BOOL;
	sWidthInUMTemp : STRING[80];
END_VAR
(**)
VAR
	p_tyLinkAlarmCurrList : REFERENCE TO ARRAY[1..c_udiAlarmCurrMax] OF tyAlarmCurr;
	p_bLinkOpConEn : REFERENCE TO BOOL;
END_VAR
```

#### Act_LinkAction.st - Change By Project
```iecst
(** 2019-04-09 **)
ACTION Act_LinkAction:

	IF p_bLinkStartupRun = TRUE THEN
	//	p_eAct ACCESS p_StartupUSOpConAct;
	ELSE
		p_eAct ACCESS ADR(eAct);

		IF p_bLinkOpConEn THEN
			bOpConRun	:= TRUE;
			bOpConStop	:= FALSE;
		ELSE
			bOpConRun	:= FALSE;
			bOpConStop	:= TRUE;
		END_IF

//		IF EDGEPOS(p_eLinkMcParamUSCommMod = McSetCommModOpCon) THEN
//			bOpConRun	:= TRUE;
//			bOpConStop	:= FALSE;
//		END_IF
//
//		IF EDGENEG(p_eLinkMcParamUSCommMod = McSetCommModOpCon) THEN
//			bOpConRun	:= FALSE;
//			bOpConStop	:= TRUE;
//		END_IF

		IF bOpConRun = TRUE THEN
			p_eAct	:= OpConActBGStartRun;

			IF (eStat = OpConActBGStartRun) AND (eStatus = Done) THEN
				p_eAct		:= OpConActIdle;
				bOpConRun	:= FALSE;
			END_IF
		END_IF

		IF bOpConStop = TRUE THEN
			p_eAct	:= OpConActBGStopRun;

			IF (eStat = OpConActBGStopRun) AND (eStatus = Done) THEN
				p_eAct		:= OpConActIdle;
				bOpConStop	:= FALSE;
			END_IF
		END_IF

	END_IF

END_ACTION
```

#### Act_Link.st - Change By Project
```iecst
(** 2019-06-04 **)
ACTION Act_Link:
	IF tyPartReceive.tyData.sTypeNo <> '' AND tyPartReceive.tyData.sTypeVar <> '' THEN
		tyPartProcessed.tyData.sTypeNo 		:= tyPartReceive.tyData.sTypeNo;
		tyPartProcessed.tyData.sTypeVar 	:= tyPartReceive.tyData.sTypeVar;
		tyPLCError.tyData.sTypeNo  			:= tyPartReceive.tyData.sTypeNo;
		tyPLCError.tyData.sTypeVar  		:= tyPartReceive.tyData.sTypeVar;
		tyPartMissing.tyData.sTypeNo  		:= tyPartReceive.tyData.sTypeNo;
		tyPartMissing.tyData.sTypeVar  		:= tyPartReceive.tyData.sTypeVar;
		tyPLCJam.tyData.sTypeNo  			:= tyPartReceive.tyData.sTypeNo;
		tyPLCJam.tyData.sTypeVar  			:= tyPartReceive.tyData.sTypeVar;
	END_IF

	IF p_bOpsTravLifULExitBrd THEN
		tyPartReceive.tyAvl.bReturnCode				:= FALSE;
	END_IF

END_ACTION
```

#### Cyclic.st - Do Not Change!!!
```iecst
(** 2019-04-21 **)
PROGRAM _CYCLIC

	IF bInitDone = FALSE THEN
		bInitDone	:= TRUE;

		Act_InitLocal;
		Act_InitGlobal;

	ELSIF bInitialDone = FALSE THEN
		IF p_bNtSettingsLoadDone = TRUE THEN
			bInitialDone	:= TRUE;

			Act_Initial;
		END_IF

	ELSE

		Act_RstErr;
		Act_LinkAction;
		Act_Action;
		Act_LinkEn;

		IF (p_bPrep = TRUE) AND (p_bEn = TRUE) AND (p_bDis = FALSE) THEN
			Act_Link;
			Act_Main;
			Act_Background;

		ELSE
			Act_Main_Disable;

			IF eStat <> OpConActIdle THEN
				eStatus	:= Done;
			ELSE
				eStatus	:= Idle;
			END_IF
		END_IF

		Act_CombineErr;
		Act_Alarm;
		Act_Alarm1;
	END_IF

END_PROGRAM
```

#### Act_InitLocal.st - Do Not Change!!!
```iecst
(** 2019-06-28 **)
ACTION Act_InitLocal:

	//Input Reference Link To Local Variable
	p_eAct ACCESS ADR(eAct);
	p_udiRstErr ACCESS ADR(udiRstErr);
	p_bPrep ACCESS ADR(bPrep);
	p_bEn ACCESS ADR(bEn);
	p_bDis ACCESS ADR(bDis);
	p_sIPAddr ACCESS ADR(sIPAddr);
	p_uiClntPort ACCESS ADR(uiClntPort); //def :0
	p_tyDTStructure ACCESS ADR(tyDTStructure);
	p_dtCurrDT ACCESS ADR(dtCurrDT);
	p_sVersion ACCESS ADR(sVersion);
	p_sRecipeNm ACCESS ADR(sRecipeNm);
	p_diWidthInUM ACCESS ADR(diWidthInUM);
	p_udiSndBffrSize ACCESS ADR(udiSndBffrSize);
	p_udiRcvBffrSize ACCESS ADR(udiRcvBffrSize);
	p_udiAliveIdleTimeInSec ACCESS ADR(udiAliveIdleTimeInSec);
	p_tConnTimeOut ACCESS ADR(tConnTimeOut);
	p_diTransferInTO ACCESS ADR(diTransferInTO);
	p_bOpsRun ACCESS ADR(bOpsRun);
	p_bInterruptSen ACCESS ADR(bInterruptSen);
	p_udiFileKeepDay ACCESS ADR(udiFileKeepDay);
	p_sProgNm ACCESS ADR(sProgNm);
	p_bNtSettingsLoadDone ACCESS ADR(bNtSettingsLoadDone);
	p_sInfoMsg ACCESS ADR(sInfoMsg);
	p_bInternalUse ACCESS ADR(bInternalUse);
	p_sInternalRcv ACCESS ADR(sInternalRcv);
	pa_tyProdRcpList ACCESS ADR(a_tyProdRcpList);
	p_tyProdRcpCurrRcp ACCESS ADR(tyProdRcpCurrRcp);

	p_tyOpConLocation ACCESS ADR (tyOpConLocation);

END_ACTION
```

#### Act_Initial.st - Do Not Change!!!
```iecst
(** 2019-04-08 **)
ACTION Act_Initial:

	//Initial
	sStatTxt	:= a_sStatText[eStat];

	fbClntConnect.udiSndBffrSize		:= p_udiSndBffrSize;
	fbClntConnect.udiRcvBffrSize		:= p_udiRcvBffrSize;
	fbClntConnect.udiAliveIdleTmInSec	:= p_udiAliveIdleTimeInSec;
	fbClntConnect.tConnectTO			:= p_tConnTimeOut;
	fbClntConnect(bEn := FALSE);

	fbRcv.udiBffrSize	:= SIZEOF(sRcv);
	fbRcv.p_BffrDest	:= ADR(sRcv);
	fbRcv(bEn := FALSE);

	fbSend.p_BffrDest	:= ADR(sSnd);
	fbSend(bEn := FALSE);

	fbClose(bEn := FALSE);

	fbParseXMLTable.p_XMLTable	:= ADR(a_tyXMLTableDataRcv);

	fbFileAppend1.sDevice	:= 'Log';
	fbFileAppend1(bEn := FALSE);

	fbFileOldDel1.sDevice			:= 'Log';
	fbFileOldDel1.sPath				:= '';
	fbFileOldDel1.sKeyword			:= p_sProgNm;
	fbFileOldDel1.udiFileKeepDay	:= p_udiFileKeepDay;
	fbFileOldDel1(bEn := FALSE);

END_ACTION
```

#### Act_Action.st - Do Not Change!!!
```iecst
(** 2019-03-25 **)
ACTION Act_Action:

	//Reset Error
	IF (eStatus = Error) AND bRstErr THEN
		p_eAct	:= OpConActIdle;
		eStat	:= OpConActIdle;
	END_IF

	//Set p_eAct
	IF eStatus = Idle OR eStatus = Busy OR eStatus = Done THEN
		eStat	:= p_eAct;
	END_IF

END_ACTION
```

#### Act_Main.st - Do Not Change!!!
```iecst
(** 2019-04-08 **)
ACTION Act_Main:

	IF eStatOld <> eStat THEN
		fbFileOldDel1(bEn := FALSE);

		sStatTxt	:= a_sStatText[eStat];

		eStatOld	:= eStat;

		eStatus		:= Busy;
	END_IF

	//Main
	CASE eStat OF

		OpConActIdle:
			eStatus	:= Idle;

		OpConActBGStartRun:
			IF eStatus = Idle OR eStatus = Busy THEN

				bRun	:= TRUE;
				bStop	:= FALSE;
				eStatus	:= Done;

			END_IF

		OpConActBGStopRun:
			IF eStatus = Idle OR eStatus = Busy THEN

				bStop	:= TRUE;
				eStatus	:= Done;

			END_IF

		OpConActDeleteOldLog:
			IF eStatus = Idle OR eStatus = Busy THEN

				eStatus	:= Busy;

				fbFileOldDel1.dtDTNow	:= p_dtCurrDT;
				fbFileOldDel1(bEn := TRUE);
				IF fbFileOldDel1.udiStatus = 0 THEN
					eStatus	:= Done;
				ELSIF fbFileOldDel1.udiStatus < 65534 THEN
					eStatus		:= Error;

					IF fbFileOldDel1.udiStatus = 1910 THEN
						udiStatus	:= 10154;	//Get Directory Info Error While Deleting Old Log
					ELSIF fbFileOldDel1.udiStatus = 1911 THEN
						udiStatus	:= 10155;	//Directory Read Error While Deleting Old Log
					ELSIF fbFileOldDel1.udiStatus = 1912 THEN
						udiStatus	:= 10156;	//File Delete Error While Deleting Old Log
					ELSE
						udiStatus	:= fbFileOldDel1.udiStatus;
					END_IF
				END_IF

			END_IF

		ELSE
			IF eStatus = Idle OR eStatus = Busy THEN
				eStatus	:= Done;
			END_IF

	END_CASE

END_ACTION
```

#### Act_Background.st - Do Not Change!!!
```iecst
(** 2019-06-10 **)
ACTION Act_Background:

	IF bRun = TRUE THEN
		IF udiTCPIdent = 0 THEN
			IF p_bInternalUse = FALSE THEN
				Act_Background_TCPConnect;

			ELSE
				udiTCPIdent	:= 1;
			END_IF

		ELSE
			IF bRstConnection = FALSE THEN
				Act_Background_TCPRcv;

//				Act_Background_NotificationRcv;
//
//				Act_Background_IllegalMsg;
//				Act_Background_ChkParamRcv;
//				Act_Background_CmpParamRcv;

//				IF bHandshakeDone = TRUE THEN
//					IF (p_tyParam.tSndAlive <> T#0s) AND (p_tyParam.tRcvAlive <> T#0s) THEN
//						IF tyServiceDescriptionRcv.tyData.tySupportedFeatures.bFeatureCheckAliveResponse = TRUE AND p_tyParam.bFeatureCheckAliveResponse = TRUE THEN
//							Act_Background_ChkAliveSendPing;
//							Act_Background_ChkAliveRcvPing;
//						ELSE
//							Act_Background_ChkAlive;
//						END_IF
//					ELSE
//						fbCheckAlive(bEn := FALSE);
//						fbCheckAliveSendPing(bEn := FALSE);
//						fbCheckAliveRcvPing(bEn := FALSE);
//					END_IF
//				END_IF

//				Act_Background_BoardAvailableChk;
				Act_Background_PLCError;
				Act_Background_Sequence;
//				Act_Background_SequenceTO;
//				Act_Background_Err;
//
//				Act_Background_ChgConfig;

				Act_Background_TCPSend;

				//				Act_Background_Log;

			ELSE //rstconnection -true
				Act_Background_TCPClose;

			END_IF

		END_IF

		Act_Background_Stop;

	END_IF

	IF EDGENEG(bRun) OR EDGENEG(udiTCPIdent = 0) THEN
		//Reset
		fbClntConnect(bEn := FALSE);

		bConnected	:= bRun;
	END_IF

	IF EDGENEG(bRun) OR EDGENEG(udiTCPIdent <> 0) THEN
		fbRcv(bEn := FALSE);
		fbSend(bEn := FALSE);
		fbClose(bEn := FALSE);

		fbFileAppend1(bEn := FALSE);

		bConnected		:= FALSE;
		bHandshakeDone	:= FALSE;
		bOverWriteSlt	:= FALSE;
		bOverWriteWidth	:= FALSE;
		bRstConnection	:= FALSE;
		bRstState		:= FALSE;

		memset(ADR(a_eMsgSend) , 0 , SIZEOF(a_eMsgSend));
		udiMsgSendBffr	:= 0;
	END_IF

	//Reset Error
	IF (eStatus1 = Error) AND bRstErr THEN
		eStatus1	:= Idle;
		udiStatus1	:= 0;

		fbClntConnect(bEn := FALSE);
		fbRcv(bEn := FALSE);
		fbSend(bEn := FALSE);
		fbClose(bEn := FALSE);

		fbFileAppend1(bEn := FALSE);

		bConnected		:= FALSE;
		bHandshakeDone	:= FALSE;
		bOverWriteSlt	:= FALSE;
		bOverWriteWidth	:= FALSE;
		bRstConnection	:= FALSE;
		bRstState		:= FALSE;

		memset(ADR(a_eMsgSend) , 0 , SIZEOF(a_eMsgSend));
		udiMsgSendBffr	:= 0;
	END_IF

END_ACTION
```

#### Act_Background_TCPConnect.st - Do Not Change!!!
```iecst
(** 2023-03-22  **)
ACTION Act_Background_TCPConnect:

	IF eStatus1 <> Error THEN

		//Connect Server
		fbClntConnect.sClntIP		:= p_sIPAddr;
		fbClntConnect.sSvrIP		:= p_sSvrIPAddr;
		fbClntConnect.uiClntPort	:= p_uiClntPort;
		fbClntConnect.uiSvrPort		:= p_uiSvrIPPort;
		fbClntConnect(bEn := TRUE);

		IF fbClntConnect.udiStatus = 0 THEN
			udiTCPIdent	:= fbClntConnect.udiTCPIdent;
			fbClntConnect(bEn := FALSE);

//		ELSIF fbClntConnect.udiStatus = 2313 THEN
//			fbClntConnect(bEn := FALSE);

//		ELSIF fbClntConnect.udiStatus = 2323 OR bConnected= FALSE THEN
//			udiStatus5	:= 10013;	//Client Connect Time Out Warning

		ELSIF fbClntConnect.udiStatus < 65534 THEN
			eStatus1	:= Error;

			IF fbClntConnect.udiStatus = 2300 THEN
				udiStatus1	:= 10000;	//Invalid Ident While Client Connecting
			ELSIF fbClntConnect.udiStatus = 2302 THEN
				udiStatus1	:= 10001;	//Setting Keep Alive Interval Time Error While Client Connecting
			ELSIF fbClntConnect.udiStatus = 2303 THEN
				udiStatus1	:= 10002;	//Setting Keep Alive Idle Time Error While Client Connecting
			ELSIF fbClntConnect.udiStatus = 2304 THEN
				udiStatus1	:= 10003;	//Setting Keep Alive Count Error While Client Connecting
			ELSIF fbClntConnect.udiStatus = 2305 THEN
				udiStatus1	:= 10004;	//Setting Keep Alive Error While Client Connecting
			ELSIF fbClntConnect.udiStatus = 2306 THEN
				udiStatus1	:= 10005;	//Setting Receive Buffer Error While Client Connecting
			ELSIF fbClntConnect.udiStatus = 2307 THEN
				udiStatus1	:= 10006;	//Setting Send Buffer Error While Client Connecting
			ELSIF fbClntConnect.udiStatus = 2308 THEN
				udiStatus1	:= 10007;	//Setting No Waiting Error While Client Connecting
			ELSIF fbClntConnect.udiStatus = 2309 THEN
				udiStatus1	:= 10008;	//TCP Open Port Error While Client Connecting
			ELSIF fbClntConnect.udiStatus = 2310 THEN
				udiStatus1	:= 10009;	//Closing TCP Error While Client Connecting
			ELSIF fbClntConnect.udiStatus = 2313 THEN
				udiStatus1	:= 10010;	//Server Connection Failed While Client Connecting
			ELSIF fbClntConnect.udiStatus = 2314 THEN
				udiStatus1	:= 10011;	//Ident In Used While Client Connecting
			ELSIF fbClntConnect.udiStatus = 2315 THEN
				udiStatus1	:= 10012;	//Connect To Server Error While Client Connecting

			ELSE
				udiStatus1	:= fbClntConnect.udiStatus;
			END_IF

		END_IF

	END_IF

END_ACTION
```

#### Act_Background_TCPRcv.st - Do Not Change!!!
```iecst
(** 2023-03-22  **)
ACTION Act_Background_TCPRcv:

	IF eStatus1 <> Error THEN

		//Receive Data
		IF p_bInternalUse = FALSE THEN
			fbRcv.udiTCPIdent	:= udiTCPIdent;
			fbRcv(bEn := TRUE);
		ELSE
			sRcv	:= p_sInternalRcv;
		END_IF

		IF (fbRcv.udiStatus = 0) OR ((p_bInternalUse = TRUE) AND (LEN(sRcv) > 0)) THEN

			fLogDTConvert(ADR(sDT) , p_dtCurrDT);
			memset(ADR(a_sLogList[udiLogCntr]) , 0 , SIZEOF(a_sLogList[udiLogCntr]));
			memcpy(ADR(a_sLogList[udiLogCntr]) + LEN(a_sLogList[udiLogCntr]) , ADR(sDT) , LEN(sDT));
			memcpy(ADR(a_sLogList[udiLogCntr]) + LEN(a_sLogList[udiLogCntr]) , ADR('$r$n') , LEN('$r$n'));
			memcpy(ADR(a_sLogList[udiLogCntr]) + LEN(a_sLogList[udiLogCntr]) , ADR('RCV_FRM_US$r$n') , LEN('RCV_FRM_US$r$n'));
			memcpy(ADR(a_sLogList[udiLogCntr]) + LEN(a_sLogList[udiLogCntr]) , ADR(sRcv) , LEN(sRcv));
			memcpy(ADR(a_sLogList[udiLogCntr]) + LEN(a_sLogList[udiLogCntr]) , ADR('$r$n$r$n') , LEN('$r$n$r$n'));

			udiLogCntr	:= udiLogCntr + 1;
			IF udiLogCntr = 11 THEN
				udiLogCntr	:= 1;
			END_IF

			fXMLConvertToTable(ADR(sRcv) , LEN(sRcv) , ADR(a_tyXMLTableDataRcv) , ADR(a_tyXMLTableDataRcv[0].sTitle) , SIZEOF(a_tyXMLTableDataRcv[0].sTitle) , ADR(a_tyXMLTableDataRcv[0].sValue) , SIZEOF(a_tyXMLTableDataRcv[0].sValue) , ADR(a_tyXMLTableDataRcv[0].uiSize) , SIZEOF(a_tyXMLTableDataRcv[0]) , SIZEOF(a_tyXMLTableDataRcv) / SIZEOF(a_tyXMLTableDataRcv[0]) , ADR(udiXMLTableWriteIdx));

			fbParseXMLTable.iTotalIdxWrite	:= UDINT_TO_INT(udiXMLTableWriteIdx);
			fbParseXMLTable;

			IF fbParseXMLTable.tyMsgType.bPartRcvRetCode = TRUE THEN
				//tyMsgTypeRcv.bCheckAlive	:= TRUE;
				tyPartReceive.tyData.iReturnCode			:= fbParseXMLTable.tyPartReceive.tyData.iReturnCode;
				tyPartReceive.tyData.sTypeNo				:= fbParseXMLTable.tyPartReceive.tyData.sTypeNo;
				tyPartReceive.tyData.sTypeVar				:= fbParseXMLTable.tyPartReceive.tyData.sTypeVar;
				tyPartReceive.tyData.sTraceTxt				:= fbParseXMLTable.tyPartReceive.tyData.sTraceTxt;
				tyPartReceive.tyAvl.bReturnCode				:= fbParseXMLTable.tyPartReceive.tyAvl.bReturnCode;
			END_IF

			IF fbParseXMLTable.tyMsgType.bPlcGrabRcv = TRUE THEN
				tyPlcGrab.tyData.iReturnCode				:= fbParseXMLTable.tyPlcGrabReceive.tyData.iReturnCode;
				tyPlcGrab.tyData.sTraceTxt					:= fbParseXMLTable.tyPlcGrabReceive.tyData.sTraceTxt;
				tyPlcGrab.tyData.sLevel						:= fbParseXMLTable.tyPlcGrabReceive.tyData.sLevel;
				tyPlcGrab.tyAvl.bReturnCode				:= fbParseXMLTable.tyPlcGrabReceive.tyAvl.bReturnCode;
			END_IF

			fbRcv(bEn := FALSE);
			memset(ADR(sRcv) , 0 , SIZEOF(sRcv));

		ELSIF (fbRcv.udiStatus = 2317) AND (p_bInternalUse = FALSE) THEN
			fbRcv(bEn := FALSE);

			memset(ADR(sRcv) , 0 , SIZEOF(sRcv));

		ELSIF (fbRcv.udiStatus = 2316) AND (p_bInternalUse = FALSE) THEN
			bRstConnection	:= TRUE;

			memset(ADR(sRcv) , 0 , SIZEOF(sRcv));

		ELSIF (fbRcv.udiStatus = 2318) AND (p_bInternalUse = FALSE) THEN
			bRstConnection	:= TRUE;

			memset(ADR(sRcv) , 0 , SIZEOF(sRcv));

		ELSIF (fbRcv.udiStatus < 65534) AND (p_bInternalUse = FALSE) THEN
			eStatus1	:= Error;

			IF fbRcv.udiStatus = 2300 THEN
				udiStatus1	:= 10014;	//Invalid Ident While Receiving Data
			ELSIF fbRcv.udiStatus = 2319 THEN
				udiStatus1	:= 10015;	//TCP Receive Data Error While Receiving Data
			ELSE
				udiStatus1	:= fbRcv.udiStatus;
			END_IF

			memset(ADR(sRcv) , 0 , SIZEOF(sRcv));

		END_IF

	END_IF

END_ACTION
```

#### Act_Background_PLCError.st - Do Not Change!!!
```iecst
 (** 2023-03-22  **)
ACTION Act_Background_PLCError:
	FOR i := 1 TO 15 DO
		IF p_tyLinkAlarmCurrList[i].eSeverity = AlmSeverityNA THEN
			IF p_tyLinkAlarmCurrList[1].eSeverity = AlmSeverityNA THEN
				memset(ADR(s1),0,SIZEOF(s1));
				memset(ADR(bMsgIssued),0,SIZEOF(bMsgIssued));
			END_IF
			EXIT;
		ELSIF p_tyLinkAlarmCurrList[i].eSeverity = AlmSeverityError THEN

			s1[i] := MID (MID(p_tyLinkAlarmCurrList[i].sMsg , LEN(p_tyLinkAlarmCurrList[i].sMsg),FIND(p_tyLinkAlarmCurrList[i].sMsg , '|')+2),LEN(p_tyLinkAlarmCurrList[i].sMsg),FIND(MID(p_tyLinkAlarmCurrList[i].sMsg , LEN(p_tyLinkAlarmCurrList[i].sMsg),FIND(p_tyLinkAlarmCurrList[i].sMsg , '|')+2) , '|')+2);
//			uiPLCErrorNo := STRING_TO_UINT (LEFT(s1[i],5));
//			sPLCErrorText := MID(s1[i],LEN(s1[i]),9);
		END_IF
//		IF s1[i] <> '' THEN
//			tyPLCError.tyData.uiErrorNo := uiPLCErrorNo;
//			tyPLCError.tyData.sErrorText := sPLCErrorText;
//		END_IF

	END_FOR

END_ACTION
```

#### Act_Background_Sequence.st - Do Not Change!!!
```iecst
 (** 2023-03-22  **)
ACTION Act_Background_Sequence:

	IF eStatus1 <> Error THEN

		IF EDGEPOS(p_tyOpsTravLifULMsgReq = OpConMsgTypePartReceived) THEN
			fOpConAddOneMsgSend(ADR(a_eMsgSend) , ADR(udiMsgSendBffr) , OpConMsgTypePartReceived);
			tyPartReceive.tyData.sIdentifier 	:= p_sOpsTravLifULBarcode;
			tyPartReceive.tyData.asName			:= 'unloader';
			tyPartReceive.tyData.asValue		:= p_tyProdRcpCurrRcp.sRcpNm;
			tyOpConEvent.tyData.uiEventId := tyOpConEvent.tyData.uiEventId +1 ;

		ELSIF EDGEPOS(p_tyOpsTravLifULMsgReq = OpConMsgTypePartProcessed)  THEN
			fOpConAddOneMsgSend(ADR(a_eMsgSend) , ADR(udiMsgSendBffr) , OpConMsgTypePartProcessed);
			tyPartProcessed.tyData.sIdentifier := p_sOpsTravLifULBarcode;
			tyPartProcessed.tyData.sValue := p_tyOpsTravLifULPartProcessItms.tyData.sValue; //[0..4]
			tyOpConEvent.tyData.uiEventId := tyOpConEvent.tyData.uiEventId +1 ;

		ELSIF EDGEPOS(p_tyOpsTravLifULMsgReq = OpConMsgTypePLCJam)  THEN
			fOpConAddOneMsgSend(ADR(a_eMsgSend) , ADR(udiMsgSendBffr) , OpConMsgTypePLCJam);
			tyOpConEvent.tyData.uiEventId := tyOpConEvent.tyData.uiEventId +1 ;

		ELSIF EDGEPOS(p_tyOpsTravLifULMsgReq = OpConMsgTypePLCJamStarted)  THEN
			fOpConAddOneMsgSend(ADR(a_eMsgSend) , ADR(udiMsgSendBffr) , OpConMsgTypePLCJamStarted);
			tyOpConEvent.tyData.uiEventId := tyOpConEvent.tyData.uiEventId +1 ;

		ELSIF EDGEPOS(p_tyOpsMagConvUL1MsgReq = OpConMsgTypePartMissingStarted) THEN
			fOpConAddOneMsgSend(ADR(a_eMsgSend) , ADR(udiMsgSendBffr) , OpConMsgTypePartMissingStarted);
			tyOpConEvent.tyData.uiEventId := tyOpConEvent.tyData.uiEventId +1 ;

		ELSIF EDGEPOS(p_tyOpsMagConvUL1MsgReq = OpConMsgTypePartMissing) THEN
			fOpConAddOneMsgSend(ADR(a_eMsgSend) , ADR(udiMsgSendBffr) , OpConMsgTypePartMissing);
			tyOpConEvent.tyData.uiEventId := tyOpConEvent.tyData.uiEventId +1 ;

		ELSIF EDGEPOS(p_tyOpsTravLifULMsgReq = OpConMsgTypePLCGrab) THEN //trav lif
			fOpConAddOneMsgSend(ADR(a_eMsgSend) , ADR(udiMsgSendBffr) , OpConMsgTypePLCGrab);
			tyOpConEvent.tyData.uiEventId := tyOpConEvent.tyData.uiEventId +1 ;
			tyPLCGrab.tyData.sValue := pas_OpsTravLifULMagEntered ;

//		ELSIF EDGEPOS(eOpConMsgReq = OpConMsgTypePLCError) THEN
//			fOpConAddOneMsgSend(ADR(a_eMsgSend) , ADR(udiMsgSendBffr) , OpConMsgTypePLCError);
//			tyOpConEvent.tyData.uiEventId := tyOpConEvent.tyData.uiEventId +1 ;
//			eOpConMsgReq := OpConMsgTypeNA;
		END_IF
		FOR i:= 1 TO 15 DO
			IF s1[i] <> '' AND bMsgIssued[i] = FALSE THEN
				eOpConMsgReq := OpConMsgTypePLCError;
				tyPLCError.tyData.uiErrorNo := STRING_TO_UINT (LEFT(s1[i],5));;
				tyPLCError.tyData.sErrorText := MID(s1[i],LEN(s1[i]),9);
				IF eOpConMsgReq = OpConMsgTypePLCError AND bMsgIssued[i] = FALSE THEN
					fOpConAddOneMsgSend(ADR(a_eMsgSend) , ADR(udiMsgSendBffr) , OpConMsgTypePLCError);
					tyOpConEvent.tyData.uiEventId := tyOpConEvent.tyData.uiEventId +1 ;
					eOpConMsgReq := OpConMsgTypeNA;
					bMsgIssued[i] := TRUE;
				END_IF
			ELSIF s1[i] = '' THEN
				EXIT;
			END_IF
		END_FOR

	END_IF

END_ACTION
```

#### Act_Background_TCPSend.st - Do Not Change!!!
```iecst
(** 2023-03-22  **)
ACTION Act_Background_TCPSend:

	//Message Send (Generate XML Message)
	IF a_eMsgSend[0] <> OpConMsgTypeNA THEN

		IF a_eMsgSend[0] = OpConMsgTypePartReceived THEN
			tyOpConEvent.tyData.sEventName := 'partReceived';
			fOpConFormPartReceive(ADR(a_tyXMLTableDataSnd) , p_tyDTStructure , tyOpConEvent, p_tyOpConLocation, tyPartReceive);
			fTableConvertToXML(ADR(sSnd) , ADR(udiSndMsgLen) , SIZEOF(sSnd) , ADR(a_tyXMLTableDataSnd) , ADR(a_tyXMLTableDataSnd[0].sTitle) , ADR(a_tyXMLTableDataSnd[0].sValue) , ADR(a_tyXMLTableDataSnd[0].uiSize) , SIZEOF(a_tyXMLTableDataSnd[0]) , 63+1);

		ELSIF a_eMsgSend[0] = OpConMsgTypePartProcessed THEN
			tyOpConEvent.tyData.sEventName := 'partProcessed';
			fOpConFormPartProcessed(ADR(a_tyXMLTableDataSnd) , p_tyDTStructure, tyOpConEvent, p_tyOpConLocation, tyPartProcessed);
			fTableConvertToXML(ADR(sSnd) , ADR(udiSndMsgLen) , SIZEOF(sSnd) , ADR(a_tyXMLTableDataSnd) , ADR(a_tyXMLTableDataSnd[0].sTitle) , ADR(a_tyXMLTableDataSnd[0].sValue) , ADR(a_tyXMLTableDataSnd[0].uiSize) , SIZEOF(a_tyXMLTableDataSnd[0]) , 123+1);

		ELSIF a_eMsgSend[0] = OpConMsgTypePLCError THEN
			tyOpConEvent.tyData.sEventName := 'plcError';
			fOpConFormPLCError(ADR(a_tyXMLTableDataSnd) , p_tyDTStructure,tyOpConEvent, p_tyOpConLocation, tyPLCError);
			fTableConvertToXML(ADR(sSnd) , ADR(udiSndMsgLen) , SIZEOF(sSnd) , ADR(a_tyXMLTableDataSnd) , ADR(a_tyXMLTableDataSnd[0].sTitle) , ADR(a_tyXMLTableDataSnd[0].sValue) , ADR(a_tyXMLTableDataSnd[0].uiSize) , SIZEOF(a_tyXMLTableDataSnd[0]) , 71+1);

		ELSIF a_eMsgSend[0] = OpConMsgTypePartMissingStarted THEN
			tyOpConEvent.tyData.sEventName := 'plcPartsMissingStarted';
			fOpConFormPartMissing(ADR(a_tyXMLTableDataSnd) , p_tyDTStructure,tyOpConEvent, p_tyOpConLocation, tyPartMissing);
			fTableConvertToXML(ADR(sSnd) , ADR(udiSndMsgLen) , SIZEOF(sSnd) , ADR(a_tyXMLTableDataSnd) , ADR(a_tyXMLTableDataSnd[0].sTitle) , ADR(a_tyXMLTableDataSnd[0].sValue) , ADR(a_tyXMLTableDataSnd[0].uiSize) , SIZEOF(a_tyXMLTableDataSnd[0]) , 59+1);

		ELSIF a_eMsgSend[0] = OpConMsgTypePartMissing THEN
			tyOpConEvent.tyData.sEventName := 'plcPartsMissing';
			fOpConFormPartMissing(ADR(a_tyXMLTableDataSnd) , p_tyDTStructure,tyOpConEvent, p_tyOpConLocation, tyPartMissing);
			fTableConvertToXML(ADR(sSnd) , ADR(udiSndMsgLen) , SIZEOF(sSnd) , ADR(a_tyXMLTableDataSnd) , ADR(a_tyXMLTableDataSnd[0].sTitle) , ADR(a_tyXMLTableDataSnd[0].sValue) , ADR(a_tyXMLTableDataSnd[0].uiSize) , SIZEOF(a_tyXMLTableDataSnd[0]) , 59+1);

		ELSIF a_eMsgSend[0] = OpConMsgTypePLCJamStarted THEN
			tyOpConEvent.tyData.sEventName := 'plcJamStarted';
			fOpConFormPLCJam(ADR(a_tyXMLTableDataSnd) , p_tyDTStructure,tyOpConEvent, p_tyOpConLocation, tyPLCJam);
			fTableConvertToXML(ADR(sSnd) , ADR(udiSndMsgLen) , SIZEOF(sSnd) , ADR(a_tyXMLTableDataSnd) , ADR(a_tyXMLTableDataSnd[0].sTitle) , ADR(a_tyXMLTableDataSnd[0].sValue) , ADR(a_tyXMLTableDataSnd[0].uiSize) , SIZEOF(a_tyXMLTableDataSnd[0]) , 57+1);

		ELSIF a_eMsgSend[0] = OpConMsgTypePLCJam THEN
			tyOpConEvent.tyData.sEventName := 'plcJam';
			fOpConFormPLCJam(ADR(a_tyXMLTableDataSnd) , p_tyDTStructure,tyOpConEvent, p_tyOpConLocation, tyPLCJam);
			fTableConvertToXML(ADR(sSnd) , ADR(udiSndMsgLen) , SIZEOF(sSnd) , ADR(a_tyXMLTableDataSnd) , ADR(a_tyXMLTableDataSnd[0].sTitle) , ADR(a_tyXMLTableDataSnd[0].sValue) , ADR(a_tyXMLTableDataSnd[0].uiSize) , SIZEOF(a_tyXMLTableDataSnd[0]) , 57+1);

		ELSIF a_eMsgSend[0] = OpConMsgTypePLCGrab THEN
			tyOpConEvent.tyData.sEventName := 'plcGrab';
			fOpConFormPLCGrab(ADR(a_tyXMLTableDataSnd) , p_tyDTStructure, tyOpConEvent,tyPLCGrab);
			fTableConvertToXML(ADR(sSnd) , ADR(udiSndMsgLen) , SIZEOF(sSnd) , ADR(a_tyXMLTableDataSnd) , ADR(a_tyXMLTableDataSnd[0].sTitle) , ADR(a_tyXMLTableDataSnd[0].sValue) , ADR(a_tyXMLTableDataSnd[0].uiSize) , SIZEOF(a_tyXMLTableDataSnd[0]) , 59+1);

		END_IF

		//Message Send
		IF p_bInternalUse = FALSE THEN
			fbSend.udiTCPIdent	:= udiTCPIdent;
			fbSend.udiSndSize	:= udiSndMsgLen;
			fbSend(bEn := TRUE);
		ELSE
			sInternalSnd	:= sSnd;
		END_IF

		IF (fbSend.udiStatus = 0) OR (p_bInternalUse = TRUE) THEN

			fLogDTConvert(ADR(sDT) , p_dtCurrDT);
			memset(ADR(a_sLogList[udiLogCntr]) , 0 , SIZEOF(a_sLogList[udiLogCntr]));
			memcpy(ADR(a_sLogList[udiLogCntr]) + LEN(a_sLogList[udiLogCntr]) , ADR(sDT) , LEN(sDT));
			memcpy(ADR(a_sLogList[udiLogCntr]) + LEN(a_sLogList[udiLogCntr]) , ADR('$r$n') , LEN('$r$n'));
			memcpy(ADR(a_sLogList[udiLogCntr]) + LEN(a_sLogList[udiLogCntr]) , ADR('SND_TO_US$r$n') , LEN('SND_TO_US$r$n'));
			memcpy(ADR(a_sLogList[udiLogCntr]) + LEN(a_sLogList[udiLogCntr]) , ADR(sSnd) , LEN(sSnd));
			memcpy(ADR(a_sLogList[udiLogCntr]) + LEN(a_sLogList[udiLogCntr]) , ADR('$r$n$r$n') , LEN('$r$n$r$n'));

			udiLogCntr	:= udiLogCntr + 1;
			IF udiLogCntr = 11 THEN
				udiLogCntr	:= 1;
			END_IF
			sSnd_0 := sSnd;

			fOpConRmvOneMsgSend(ADR(a_eMsgSend) , ADR(udiMsgSendBffr));

			fbSend(bEn := FALSE);

		ELSIF (fbSend.udiStatus = 2321) AND (p_bInternalUse = FALSE) THEN
			bRstConnection	:= TRUE;

		ELSIF (fbSend.udiStatus < 65534) AND (p_bInternalUse = FALSE) THEN
			eStatus1	:= Error;

			IF fbSend.udiStatus = 2300 THEN
				udiStatus1	:= 10143;	//Invalid Ident While Sending Data
			ELSIF fbSend.udiStatus = 2320 THEN
				udiStatus1	:= 10144;	//TCP Retry Send Data Error While Sending Data
			ELSIF fbSend.udiStatus = 2322 THEN
				udiStatus1	:= 10145;	//TCP Send Data Error
			ELSE
				udiStatus1	:= fbSend.udiStatus;
			END_IF

		END_IF

	END_IF

	IF bTestEn THEN
		fbFileFullWrite_0(bEn := TRUE, sDevice := 'Log', sFile := 'OpCon_Send.xml', udiOffset := 0, p_Src := ADR(sSnd_0), udiLen := SIZEOF(sSnd_0), udiOption := 0);
		IF fbFileFullWrite_0.udiStatus = 0 THEN
			fbFileFullWrite_0(bEn := FALSE);
			bTestEn := FALSE;
		END_IF

	ELSE
		fbFileFullWrite_0(bEn := FALSE);
	END_IF

END_ACTION
```

#### Act_Background_TCPClose.st - Do Not Change!!!
```iecst
(** 2023-03-22  **)
ACTION Act_Background_TCPClose:

	//Close TCP Connection
	IF p_bInternalUse = FALSE THEN
		fbClose.udiTCPIdent	:= udiTCPIdent;
		fbClose(bEn := TRUE);

		IF fbClose.udiStatus = 0 THEN
			udiTCPIdent	:= 0;
			fbClose(bEn := FALSE);

		ELSIF fbClose.udiStatus < 65534 THEN
			udiTCPIdent	:= 0;
			eStatus1	:= Error;

			IF fbClose.udiStatus = 2300 THEN
				udiStatus1	:= 10146;	//Invalid Ident While Closing TCP
			ELSIF fbClose.udiStatus = 2310 THEN
				udiStatus1	:= 10147;	//Closing TCP Error
			ELSE
				udiStatus1	:= fbClose.udiStatus;
			END_IF

		END_IF

	ELSE
		udiTCPIdent	:= 0;

	END_IF

END_ACTION
```

#### Act_Background_Stop.st - Do Not Change!!!
```iecst
(** 2019-03-15 **)
ACTION Act_Background_Stop:

	IF bStop = TRUE THEN

		IF a_eMsgSend[0] = OpConMsgTypeNA THEN

			bRstConnection	:= TRUE;

			IF udiTCPIdent = 0 THEN

				bRun	:= FALSE;

			END_IF

		END_IF

	END_IF

END_ACTION
```

#### Act_Background_Log.st - Do Not Change!!!
```iecst
(** 2019-05-01 **)
ACTION Act_Background_Log:

//	IF eStatus3 <> Error THEN
//
//		IF udiWriteLogCntr <> udiLogCntr THEN
//
//			CASE iWriteLogStep OF
//
//				0:
//					dtCurrDTTemp			:= p_dtCurrDT;
//					fbFileAppend1.sFile		:= DT_TO_STRING(dtCurrDTTemp);
//					fbFileAppend1.sFile		:= MID(fbFileAppend1.sFile , 10 , 4);
//					fbFileAppend1.sFile		:= CONCAT('_' , fbFileAppend1.sFile);
//					fbFileAppend1.sFile		:= CONCAT(p_sProgNm , fbFileAppend1.sFile);
//					fbFileAppend1.sFile		:= CONCAT(fbFileAppend1.sFile , '.dat');
//
//					fbFileAppend1.p_Src		:= ADR(a_sLogList[udiWriteLogCntr]);
//					fbFileAppend1.udiLen	:= LEN(a_sLogList[udiWriteLogCntr]);
//
//					iWriteLogStep	:= 1;
//
//				1:
//					fbFileAppend1(bEn := TRUE);
//					IF fbFileAppend1.udiStatus = 0 THEN
//						fbFileAppend1(bEn := FALSE);
//
//						udiWriteLogCntr	:= udiWriteLogCntr + 1;
//						IF udiWriteLogCntr = 11 THEN
//							udiWriteLogCntr	:= 1;
//						END_IF
//
//						iWriteLogStep	:= 0;
//
//					ELSIF fbFileAppend1.udiStatus < 65534 THEN
//						eStatus3	:= Error;
//
//						IF fbFileAppend1.udiStatus = 1900 THEN
//							udiStatus3	:= 10148;	//File Open Error While Writing Log
//						ELSIF fbFileAppend1.udiStatus = 1901 THEN
//							udiStatus3	:= 10149;	//File Create Error While Writing Log
//						ELSIF fbFileAppend1.udiStatus = 1913 THEN
//							udiStatus3	:= 10150;	//Get File Info Error While Writing Log
//						ELSIF fbFileAppend1.udiStatus = 1903 THEN
//							udiStatus3	:= 10151;	//File Write Error While Writing Log
//						ELSIF fbFileAppend1.udiStatus = 1904 THEN
//							udiStatus3	:= 10152;	//File Close Error While Writing Log
//						ELSIF fbFileAppend1.udiStatus = 1914 THEN
//							udiStatus3	:= 10153;	//Directory Does Not Exist While Writing Log
//						ELSE
//							udiStatus3	:= fbFileAppend1.udiStatus;
//						END_IF
//
//						iWriteLogStep	:= 0;
//
//					END_IF
//
//			END_CASE
//
//		END_IF
//
//	END_IF

END_ACTION
```

#### Act_Background_Err.st - Do Not Change!!!
```iecst
(** 2019-03-15 **)
ACTION Act_Background_Err:

END_ACTION
```

#### Act_Main_Disable.st - Do Not Change!!!
```iecst
(** 2019-03-15 **)
ACTION Act_Main_Disable:

	bConnected		:= FALSE;
	bHandshakeDone	:= FALSE;
	bOverWriteSlt	:= FALSE;
	bOverWriteWidth	:= FALSE;

END_ACTION
```

#### Act_CombineErr.st - Do Not Change!!!
```iecst
(** 2019-03-15 **)
ACTION Act_CombineErr:

	//Combine Error
	IF eStatus = Error OR eStatus1 = Error THEN
		eMainStatus	:= Error;
	ELSE
		eMainStatus	:= eStatus;
	END_IF

END_ACTION
```

#### Act_Alarm.st - Do Not Change!!!
```iecst
(** 2019-03-25 **)
ACTION Act_Alarm:

	//Error
	IF EDGEPOS(eStatus = Error) THEN

		tyAlmData.sProgNm		:= p_sProgNm;
		tyAlmData.udiCode		:= udiStatus;
		tyAlmData.eSeverity		:= AlmSeverityError;
		tyAlmData.udiRunTime	:= tyAlmData.udiRunTime + 1;

		//Get Error Message
		IF tyAlmData.udiCode < 10000 OR tyAlmData.udiCode > 10199 THEN
			tyAlmData.sAlmMsg	:= 'Unknown';
			tyAlmData.sRcyMsg	:= 'Unknown';
		ELSE
			tyAlmData.sAlmMsg	:= a_tyAlmText[tyAlmData.udiCode].sAlmText;
			tyAlmData.sRcyMsg	:= a_tyAlmText[tyAlmData.udiCode].sRcyText;
		END_IF

		sStatTxt	:= tyAlmData.sAlmMsg;

	ELSIF bRstErr AND (tyAlmData.udiCode <> 0) THEN

		tyAlmData.udiCode	:= 0;
		tyAlmData.eSeverity	:= AlmSeverityNA;
		tyAlmData.sAlmMsg	:= '';
		tyAlmData.sRcyMsg	:= '';

		sStatTxt	:= a_sStatText[eStat];

	END_IF

END_ACTION
```

#### Act_Alarm1.st - Do Not Change!!!
```iecst
(** 2019-03-25 **)
ACTION Act_Alarm1:

	//Error
	IF EDGEPOS(eStatus1 = Error) THEN

		tyAlmData1.sProgNm		:= p_sProgNm;
		tyAlmData1.udiCode		:= udiStatus1;
		tyAlmData1.eSeverity	:= AlmSeverityError;
		tyAlmData1.udiRunTime	:= tyAlmData1.udiRunTime + 1;

		//Get Error Message
		IF tyAlmData1.udiCode < 10000 OR tyAlmData1.udiCode > 10199 THEN
			tyAlmData1.sAlmMsg	:= 'Unknown';
			tyAlmData1.sRcyMsg	:= 'Unknown';
		ELSE
			tyAlmData1.sAlmMsg	:= a_tyAlmText[tyAlmData1.udiCode].sAlmText;
			tyAlmData1.sRcyMsg	:= a_tyAlmText[tyAlmData1.udiCode].sRcyText;
		END_IF

		sStatTxt	:= tyAlmData1.sAlmMsg;

	ELSIF bRstErr AND (tyAlmData1.udiCode <> 0) THEN

		tyAlmData1.udiCode		:= 0;
		tyAlmData1.eSeverity	:= AlmSeverityNA;
		tyAlmData1.sAlmMsg		:= '';
		tyAlmData1.sRcyMsg		:= '';

		sStatTxt	:= a_sStatText[eStat];

	END_IF

END_ACTION
```

#### InputRef.var - Do Not Change!!!
```iecst
(*2019-06-28*)
(**)
(*General*)
VAR
	p_eAct : REFERENCE TO eOpConAction;
	p_udiRstErr : REFERENCE TO UDINT;
	p_bPrep : REFERENCE TO BOOL;
	p_bEn : REFERENCE TO BOOL;
	p_bDis : REFERENCE TO BOOL;
END_VAR
(**)
(*Configuration*)
VAR
	p_sIPAddr : REFERENCE TO STRING[15];
	p_uiClntPort : REFERENCE TO USINT;
	p_sSvrIPAddr : REFERENCE TO STRING[15];
	p_uiSvrIPPort : REFERENCE TO UINT;
	p_tyDTStructure : REFERENCE TO DTStructure;
	p_dtCurrDT : REFERENCE TO DATE_AND_TIME;
END_VAR
(**)
(*Input*)
VAR
	p_sVersion : REFERENCE TO STRING[7];
	p_sRecipeNm : REFERENCE TO STRING[254];
	p_diWidthInUM : REFERENCE TO DINT;
	p_udiSndBffrSize : REFERENCE TO UDINT;
	p_udiRcvBffrSize : REFERENCE TO UDINT;
	p_udiAliveIdleTimeInSec : REFERENCE TO UDINT;
	p_tConnTimeOut : REFERENCE TO TIME;
	p_diTransferInTO : REFERENCE TO DINT;
	p_bOpsRun : REFERENCE TO BOOL;
	p_bInterruptSen : REFERENCE TO BOOL;
	p_udiFileKeepDay : REFERENCE TO UDINT;
	p_sProgNm : REFERENCE TO STRING[15];
	p_bNtSettingsLoadDone : REFERENCE TO BOOL;
	p_sInfoMsg : REFERENCE TO STRING[200];
	p_bInternalUse : REFERENCE TO BOOL;
	p_sInternalRcv : REFERENCE TO STRING[65535];
	pa_tyProdRcpList : REFERENCE TO ARRAY[1..c_udiProdRcpMax] OF tyProdRcpParam;
	p_tyProdRcpCurrRcp : REFERENCE TO tyProdRcpParam;
	p_tyOpConLocation : REFERENCE TO tyLocationParam;
	p_bOpsTravLifULExitBrd : REFERENCE TO BOOL;
	p_tyOpsTravLifULMsgReq : REFERENCE TO eOpConMsgType;
	p_tyOpsMagConvUL1MsgReq : REFERENCE TO eOpConMsgType;
	p_tyOpsTravLifULPartProcessItms : REFERENCE TO tyOpConPartProcessed;
	pas_OpsTravLifULMagEntered : REFERENCE TO ARRAY[0..4] OF STRING[10];
	pa_OpsTravLifULMagEntered : REFERENCE TO ARRAY[1..4] OF BOOL;
	p_sOpsTravLifULBarcode : REFERENCE TO STRING[80];
END_VAR
```

#### Local.var - Do Not Change!!!
```iecst
(*2019-06-28*)
(**)
(*Local Action, State & Status*)
VAR
	eAct : eOpConAction := OpConActIdle;
	eStat : eOpConAction := OpConActIdle;
	eStatOld : eOpConAction := OpConActIdle;
	eMainStatus : eFBStatus := Idle;
	eStatus : eFBStatus := Idle;
	eStatus1 : eFBStatus := Idle;
	udiStatus : UDINT := 0;
	udiStatus1 : UDINT := 0;
	sStatTxt : STRING[200] := '';
	a_sStatText : ARRAY[0..50] OF STRING[200] := ['Idling','Background Starting Operations','Background Stopping Operations','Deleting Old Log File','Creating Directory','Writing Retain File','Reading Retain File','Saving Configuration',43('')];
END_VAR
(**)
(*Local Alarm*)
VAR
	tyAlmData : tyAlmDat;
	tyAlmData1 : tyAlmDat;
	tyInfoData : tyAlmDat;
	a_tyAlmText : ARRAY[10000..10199] OF tyAlmTxt := [(sAlmText:='Invalid Ident While Client Connecting',sRcyText:='Problem Occurred In The TCP/IP Connection. Check The Connection And Try To Reconnect.'),(sAlmText:='Setting Keep Alive Interval Time Error While Client Connecting',sRcyText:='Unable To Establish Connection Between Machine. Check For Setting And Resume Operation.'),(sAlmText:='Setting Keep Alive Idle Time Error While Client Connecting',sRcyText:='Unable To Establish Connection Between Machine. Check For Setting And Resume Operation.'),(sAlmText:='Setting Keep Alive Count Error While Client Connecting',sRcyText:='Unable To Establish Connection Between Machine. Check For Setting And Resume Operation.'),(sAlmText:='Setting Keep Alive Error While Client Connecting',sRcyText:='Unable To Establish Connection Between Machine. Check For Setting And Resume Operation.'),(sAlmText:='Setting Receive Buffer Error While Client Connecting',sRcyText:='Unable To Establish Connection Between Machine. Check For Setting And Resume Operation.'),(sAlmText:='Setting Send Buffer Error While Client Connecting',sRcyText:='Unable To Establish Connection Between Machine. Check For Setting And Resume Operation.'),(sAlmText:='Setting No Waiting Error While Client Connecting',sRcyText:='Unable To Establish Connection Between Machine. Check For Setting And Resume Operation.'),(sAlmText:='TCP Open Port Error While Client Connecting',sRcyText:='Problem Occurred In The TCP/IP Connection. Check The Connection And Try To Reconnect.'),(sAlmText:='Closing TCP Error While Client Connecting',sRcyText:='Problem Occurred In The TCP/IP Connection. Check The Connection And Try To Reconnect.'),(sAlmText:='Server Connection Failed While Client Connecting',sRcyText:='There Was A Problem Connecting To The Server. The Server May Not Exist or It is Unavailable At This Time. Check The Connection and Try Again.'),(sAlmText:='Ident In Used While Client Connecting',sRcyText:='Problem Occurred In The TCP/IP Connection. Check The Connection And Reconnect.'),(sAlmText:='Connect To Server Error While Client Connecting',sRcyText:='There Was A Problem Connecting To The Server. The Server May Not Exist or It is Unavailable At This Time. Check The Connection and Try Again.'),(sAlmText:='US Hermes Connection Lost',sRcyText:='Please Check Network Connection'),(sAlmText:='Invalid Ident While Receiving Data',sRcyText:='Problem Occurred In The TCP/IP Connection. Check The Connection And Try To Reconnect.'),(sAlmText:='TCP Receive Data Error While Receiving Data',sRcyText:='Problem Occurred In The TCP/IP Connection. Check The Connection And Try To Reconnect.'),(sAlmText:='Receive ServiceDescription While Upstream In Not Connected State',sRcyText:='Receive Illegal Message.'),(sAlmText:='Receive BoardAvailable While Upstream In Not Connected State',sRcyText:='Receive Illegal Message.'),(sAlmText:='Receive RevokeBoardAvailable While Upstream In Not Connected State',sRcyText:='Receive Illegal Message.'),(sAlmText:='Receive MachineReady While Upstream In Not Connected State',sRcyText:='Receive Illegal Message.'),(sAlmText:='Receive RevokeMachineReady While Upstream In Not Connected State',sRcyText:='Receive Illegal Message.'),(sAlmText:='Receive StartTransport While Upstream In Not Connected State',sRcyText:='Receive Illegal Message.'),(sAlmText:='Receive StopTransport While Upstream In Not Connected State',sRcyText:='Receive Illegal Message.'),(sAlmText:='Receive TransportFinished While Upstream In Not Connected State',sRcyText:='Receive Illegal Message.'),(sAlmText:='Receive BoardForecast While Upstream In Not Connected State',sRcyText:='Receive Illegal Message.'),(sAlmText:='Receive BoardAvailable While Upstream In Service Description State',sRcyText:='Receive Illegal Message.'),(sAlmText:='Receive RevokeBoardAvailable While Upstream In Service Description State',sRcyText:='Receive Illegal Message.'),(sAlmText:='Receive MachineReady While Upstream In Service Description State',sRcyText:='Receive Illegal Message.'),(sAlmText:='Receive RevokeMachineReady While Upstream In Service Description State',sRcyText:='Receive Illegal Message.'),(sAlmText:='Receive StartTransport While Upstream In Service Description State',sRcyText:='Receive Illegal Message.'),(sAlmText:='Receive StopTransport While Upstream In Service Description State',sRcyText:='Receive Illegal Message.'),(sAlmText:='Receive TransportFinished While Upstream In Service Description State',sRcyText:='Receive Illegal Message.'),(sAlmText:='Receive BoardForecast While Upstream In Service Description State',sRcyText:='Receive Illegal Message.'),(sAlmText:='Receive ServiceDescription While Upstream In Not Available Not Ready State',sRcyText:='Receive Illegal Message.'),(sAlmText:='Receive RevokeBoardAvailable While Upstream In Not Available Not Ready State',sRcyText:='Receive Illegal Message.'),(sAlmText:='Receive MachineReady While Upstream In Not Available Not Ready State',sRcyText:='Receive Illegal Message.'),(sAlmText:='Receive RevokeMachineReady While Upstream In Not Available Not Ready State',sRcyText:='Receive Illegal Message.'),(sAlmText:='Receive StartTransport While Upstream In Not Available Not Ready State',sRcyText:='Receive Illegal Message.'),(sAlmText:='Receive StopTransport While Upstream In Not Available Not Ready State',sRcyText:='Receive Illegal Message.'),(sAlmText:='Receive TransportFinished While Upstream In Not Available Not Ready State',sRcyText:='Receive Illegal Message.'),(sAlmText:='Receive ServiceDescription While Upstream In Board Available State',sRcyText:='Receive Illegal Message.'),(sAlmText:='Receive BoardAvailable While Upstream In Board Available State',sRcyText:='Receive Illegal Message.'),(sAlmText:='Receive MachineReady While Upstream In Board Available State',sRcyText:='Receive Illegal Message.'),(sAlmText:='Receive RevokeMachineReady While Upstream In Board Available State',sRcyText:='Receive Illegal Message.'),(sAlmText:='Receive StartTransport While Upstream In Board Available State',sRcyText:='Receive Illegal Message.'),(sAlmText:='Receive StopTransport While Upstream In Board Available State',sRcyText:='Receive Illegal Message.'),(sAlmText:='Receive TransportFinished While Upstream In Board Available State',sRcyText:='Receive Illegal Message.'),(sAlmText:='Receive BoardForecast While Upstream In Board Available State',sRcyText:='Receive Illegal Message.'),(sAlmText:='Receive ServiceDescription While Upstream In Machine Ready State',sRcyText:='Receive Illegal Message.'),(sAlmText:='Receive RevokeBoardAvailable While Upstream In Machine Ready State',sRcyText:='Receive Illegal Message.'),(sAlmText:='Receive MachineReady While Upstream In Machine Ready State',sRcyText:='Receive Illegal Message.'),(sAlmText:='Receive RevokeMachineReady While Upstream In Machine Ready State',sRcyText:='Receive Illegal Message.'),(sAlmText:='Receive StartTransport While Upstream In Machine Ready State',sRcyText:='Receive Illegal Message.'),(sAlmText:='Receive StopTransport While Upstream In Machine Ready State',sRcyText:='Receive Illegal Message.'),(sAlmText:='Receive TransportFinished While Upstream In Machine Ready State',sRcyText:='Receive Illegal Message.'),(sAlmText:='Receive ServiceDescription While Upstream In Available And Ready State',sRcyText:='Receive Illegal Message.'),(sAlmText:='Receive BoardAvailable While Upstream In Available And Ready State',sRcyText:='Receive Illegal Message.'),(sAlmText:='Receive MachineReady While Upstream In Available And Ready State',sRcyText:='Receive Illegal Message.'),(sAlmText:='Receive RevokeMachineReady While Upstream In Available And Ready State',sRcyText:='Receive Illegal Message.'),(sAlmText:='Receive StartTransport While Upstream In Available And Ready State',sRcyText:='Receive Illegal Message.'),(sAlmText:='Receive StopTransport While Upstream In Available And Ready State',sRcyText:='Receive Illegal Message.'),(sAlmText:='Receive TransportFinished While Upstream In Available And Ready State',sRcyText:='Receive Illegal Message.'),(sAlmText:='Receive BoardForecast While Upstream In Available And Ready State',sRcyText:='Receive Illegal Message.'),(sAlmText:='Receive ServiceDescription While Upstream In Transporting State',sRcyText:='Receive Illegal Message.'),(sAlmText:='Receive Twice Board Available While Upstream In Transporting State',sRcyText:='Receive Illegal Message.'),(sAlmText:='Receive RevokeBoardAvailable Without BoardAvailable While Upstream In Transporting State',sRcyText:='Receive Illegal Message.'),(sAlmText:='Receive MachineReady While Upstream In Transporting State',sRcyText:='Receive Illegal Message.'),(sAlmText:='Receive RevokeMachineReady While Upstream In Transporting State',sRcyText:='Receive Illegal Message.'),(sAlmText:='Receive StartTransport While Upstream In Transporting State',sRcyText:='Receive Illegal Message.'),(sAlmText:='Receive StopTransport While Upstream In Transporting State',sRcyText:='Receive Illegal Message.'),(sAlmText:='Receive ServiceDescription While Upstream In Transport Finished State',sRcyText:='Receive Illegal Message.'),(sAlmText:='Receive BoardAvailable While Upstream In Transport Finished State',sRcyText:='Receive Illegal Message.'),(sAlmText:='Receive RevokeBoardAvailable While UpstreamWhile Upstream In Transport Finished State',sRcyText:='Receive Illegal Message.'),(sAlmText:='Receive MachineReady While Upstream In Transport Finished State',sRcyText:='Receive Illegal Message.'),(sAlmText:='Receive RevokeMachineReady While Upstream In Transport Finished State',sRcyText:='Receive Illegal Message.'),(sAlmText:='Receive StartTransport While Upstream In Transport Finished State',sRcyText:='Receive Illegal Message.'),(sAlmText:='Receive TransportFinished While Upstream In Transport Finished State',sRcyText:='Receive Illegal Message.'),(sAlmText:='Receive StopTransport While Upstream In Transport Finished State',sRcyText:='Receive Illegal Message.'),(sAlmText:='Receive BoardForecast While Upstream In Transport Finished State',sRcyText:='Receive Illegal Message.'),(sAlmText:='Receive ServiceDescription While Upstream In Transport Stopped State',sRcyText:='Receive Illegal Message.'),(sAlmText:='Receive Twice Board Available While Upstream In Transport Stopped State',sRcyText:='Receive Illegal Message.'),(sAlmText:='Receive RevokeBoardAvailable Without BoardAvailable While Upstream In Transport Stopped State',sRcyText:='Receive Illegal Message.'),(sAlmText:='Receive MachineReady While Upstream In Transport Stopped State',sRcyText:='Receive Illegal Message.'),(sAlmText:='Receive RevokeMachineReady While Upstream In Transport Stopped State',sRcyText:='Receive Illegal Message.'),(sAlmText:='Receive StartTransport While Upstream In Transport Stopped State',sRcyText:='Receive Illegal Message.'),(sAlmText:='Receive StopTransport While Upstream In Transport Stopped State',sRcyText:='Receive Illegal Message.'),(sAlmText:='LaneId Mismatch While Checking Service Description',sRcyText:='The LaneId Value Does Not Match. Change The Value And Resend The Value.'),(sAlmText:='MachineId Missing While Checking Service Description',sRcyText:='Missing Input Value For MachineId. Fill Up The Value And Resend.'),(sAlmText:='LandId Out Of Range While Checking Service Description',sRcyText:='LaneId Does Not Fall Within The Expected Range.'),(sAlmText:='LandId Missing While Checking Service Description',sRcyText:='Missing Input Value For LaneId. Fill Up The Value And Resend.'),(sAlmText:='Version Missing While Checking Service Description',sRcyText:='Missing Input Value For Version. Fill Up The Value And Resend.'),(sAlmText:='SupportedFeatures Missing While Checking Service Description',sRcyText:='Missing Input Value For SupportedFeatures. Fill Up The Value And Resend.'),(sAlmText:='NotificationCode Out Of Range While Checking Notification',sRcyText:='NotificationCode Does Not Fall Within The Expected Range.'),(sAlmText:='NotificationCode Missing While Checking Notification',sRcyText:='Missing Input Value For NotificationCode. Fill Up The Value And Resend.'),(sAlmText:='Severity Missing While Checking Notification',sRcyText:='Missing Input Value For Severity. Fill Up The Value And Resend.'),(sAlmText:='Description Missing While Checking Notification',sRcyText:='Missing Input Value For Description. Fill Up The Value And Resend.'),(sAlmText:='BoardId Missing While Checking Board Available',sRcyText:='Missing Input Value For BoardId. Fill Up The Value And Resend.'),(sAlmText:='BoardIdCreatedBy Missing While Checking Board Available',sRcyText:='Missing Input Value For BoardIdCreatedBy. Fill Up The Value And Resend.'),(sAlmText:='FailedBoard Missing While Checking Board Available',sRcyText:='Missing Input Value For FailedBoard. Fill Up The Value And Resend.'),(sAlmText:='FlippedBoard Missing While Checking Board Available',sRcyText:='Missing Input Value For FlippedBoard. Fill Up The Value And Resend.'),(sAlmText:='TransferState Missing While Checking Transport Finished',sRcyText:='Missing Input Value For TransferState. Fill Up The Value And Resend.'),(sAlmText:='BoardId Missing While Checking Transport Finished',sRcyText:='Missing Input Value For BoardId. Fill Up The Value And Resend.'),(sAlmText:='FailedBoard Missing While Checking Board Forecast',sRcyText:='Missing Input Value For FailedBoard. Fill Up The Value And Resend.'),(sAlmText:='FlippedBoard Missing While Checking Board Forecast',sRcyText:='Missing Input Value For FlippedBoard. Fill Up The Value And Resend.'),(sAlmText:='BoardId Mismatch While Checking Start Transport & Transport Finished',sRcyText:='The BoardId Value Does Not Match. Change The Value And Resend The Value.'),(sAlmText:='BoardId Missing While Checking Start Transport & Transport Finished',sRcyText:='Missing Input Value For BoardId. Fill Up The Value And Resend.'),(sAlmText:='Service Description Interchange Time Out',sRcyText:='Timeout Expired Before Operation Completed. Reset And Resume Operation.'),(sAlmText:='Transport Time Out',sRcyText:='Timeout Expired Before Operation Completed. Reset And Resume Operation.'),(sAlmText:='Input First Slot Is Invalid',sRcyText:='Invalid Input Value.'),(sAlmText:='Input Last Slot Is Invalid',sRcyText:='Invalid Input Value.'),(sAlmText:='Input Pitch Is Invalid',sRcyText:='Invalid Input Value.'),(sAlmText:='Input Slot To Slot Distance Is Invalid',sRcyText:='Invalid Input Value.'),(sAlmText:='Input Total Slot Is Invalid',sRcyText:='Invalid Input Value.'),(sAlmText:='Input Thickness Is Invalid',sRcyText:='Invalid Input Value.'),(sAlmText:='Input Top Clearance Height Is Invalid',sRcyText:='Invalid Input Value.'),(sAlmText:='Input Bottom Clearance Height Is Invalid',sRcyText:='Invalid Input Value.'),(sAlmText:='Recipe First Slot Value & Board Available Data Not Match With Same Product Type Id',sRcyText:='The Recipe First Slot Value & Board Available Data Value Does Not Match With Product Type ID. Change The Value And Resend The Value.'),(sAlmText:='Recipe Last Slot Value & Board Available Data Not Match With Same Product Type Id',sRcyText:='The Recipe Last Slot Value & Board Available Data Value Does Not Match With Product Type ID. Change The Value And Resend The Value.'),(sAlmText:='Recipe Pitch Value & Board Available Data Not Match With Same Product Type Id',sRcyText:='The Recipe Pitch Value & Board Available Data Value Does Not Match With Product Type ID. Change The Value And Resend The Value.'),(sAlmText:='Width Different With Same Product Type Id',sRcyText:='Width Does Not Match With Product Type ID. Change The Value And Resend The Value.'),(sAlmText:='Input First Slot Is Invalid',sRcyText:='Invalid Input Value.'),(sAlmText:='Input Last Slot Is Invalid',sRcyText:='Invalid Input Value.'),(sAlmText:='Input Pitch Is Invalid',sRcyText:='Invalid Input Value.'),(sAlmText:='Input Slot To Slot Distance Is Invalid',sRcyText:='Invalid Input Value.'),(sAlmText:='Input Total Slot Is Invalid',sRcyText:='Invalid Input Value.'),(sAlmText:='Input Thickness Is Invalid',sRcyText:='Invalid Input Value.'),(sAlmText:='Input Top Clearance Height Is Invalid',sRcyText:='Invalid Input Value.'),(sAlmText:='Input Bottom Clearance Height Is Invalid',sRcyText:='Invalid Input Value.'),(sAlmText:='Recipe First Slot Value & Board Available Data Not Match With Same Product Type Id',sRcyText:='The Recipe First Slot Value & Board Available Data Value Does Not Match With Product Type ID. Change The Value And Resend The Value.'),(sAlmText:='Recipe Last Slot Value & Board Available Data Not Match With Same Product Type Id',sRcyText:='The Recipe Last Slot Value & Board Available Data Value Does Not Match With Product Type ID. Change The Value And Resend The Value.'),(sAlmText:='Recipe Pitch Value & Board Available Data Not Match With Same Product Type Id',sRcyText:='The Recipe Pitch Value & Board Available Data Value Does Not Match With Product Type ID. Change The Value And Resend The Value.'),(sAlmText:='Width Different With Same Product Type Id',sRcyText:='Width Does Not Match With Product Type ID. Change The Value And Resend The Value.'),(sAlmText:='Check Alive Time Out',sRcyText:='Timeout Expired Before Operation Completed. Reset And Resume Operation.'),(sAlmText:='Waiting Check Alive Time Out',sRcyText:='Timeout Expired Before Operation Completed. Reset And Resume Operation.'),(sAlmText:='Check Alive Id Mismatch',sRcyText:='The Check Alive Id Value Does Not Match. Change The Value And Resend The Value.'),(sAlmText:='Board Available Request To Send From Upstream Hermes',sRcyText:='Sending Illegal Message.'),(sAlmText:='Revoke Board Available Request To Send From Upstream Hermes',sRcyText:='Sending Illegal Message.'),(sAlmText:='Transport Finished Request To Send From Upstream Hermes',sRcyText:='Sending Illegal Message.'),(sAlmText:='Set Configuration Request To Send From Upstream Hermes',sRcyText:='Sending Illegal Message.'),(sAlmText:='Get Configuration Request To Send From Upstream Hermes',sRcyText:='Sending Illegal Message.'),(sAlmText:='Current Configuration Request To Send From Upstream Hermes',sRcyText:='Sending Illegal Message.'),(sAlmText:='Board Forecast Request To Send From Upstream Hermes',sRcyText:='Sending Illegal Message.'),(sAlmText:='Send Board Info Request To Send From Upstream Hermes',sRcyText:='Sending Illegal Message.'),(sAlmText:='Invalid Ident While Sending Data',sRcyText:='Invalid Ident Value.'),(sAlmText:='TCP Retry Send Data Error While Sending Data',sRcyText:='Problem Occurred In The TCP/IP Connection. Check The Connection And Try To Reconnect.'),(sAlmText:='TCP Send Data Error',sRcyText:='Problem Occurred In The TCP/IP Connection. Check The Connection And Try To Reconnect.'),(sAlmText:='Invalid Ident While Closing TCP',sRcyText:='Invalid Ident Value.'),(sAlmText:='Closing TCP Error',sRcyText:='Problem Occurred In The TCP/IP Connection. Check The Connection And Try To Reconnect.'),(sAlmText:='File Open Error While Writing Log',sRcyText:='An Error Was Encountered While Trying To Open File. Please Contact Nutek For A Possible Solution.'),(sAlmText:='File Create Error While Writing Log',sRcyText:='An Error Was Encountered While Trying To Create File. Please Contact Nutek For A Possible Solution.'),(sAlmText:='Get File Info Error While Writing Log',sRcyText:='An Error Was Encountered While Getting File Info. Please Contact Nutek For A Possible Solution.'),(sAlmText:='File Write Error While Writing Log',sRcyText:='An Error Was Encountered While Trying To Write File. Please Contact Nutek For A Possible Solution.'),(sAlmText:='File Close Error While Writing Log',sRcyText:='An Error Was Encountered While Trying To Close File. Please Contact Nutek For A Possible Solution.'),(sAlmText:='Directory Does Not Exist While Writing Log',sRcyText:='The Directory Does Not Exist.Please Contact Nutek For A Possible Solution.'),(sAlmText:='Get Directory Info Error While Deleting Old Log',sRcyText:='An Error Was Encountered While Getting Directory Info. Please Contact Nutek For A Possible Solution.'),(sAlmText:='Directory Read Error While Deleting Old Log',sRcyText:='An Error Was Encountered While Reading Directory. Please Contact Nutek For A Possible Solution.'),(sAlmText:='File Delete Error While Deleting Old Log',sRcyText:='An Error Was Encountered While Trying To Delete File. Please Contact Nutek For A Possible Solution.'),(sAlmText:='Board Jam At Sensor After Transfer Interrupted',sRcyText:='Push Back Board To Upstream Machine'),(sAlmText:='Product Type Id Not Receive From Upstream',sRcyText:='Check Upstream Machine Whether Product Type Id Is Used.'),10((0)),(sAlmText:='New Recipe Not Found In Product Recipe List',sRcyText:='Create New Recipe In Product Setting.'),30((0))];
END_VAR
(**)
(*Local Output*)
VAR
	a_tyXMLTableDataBrdAvl : ARRAY[0..200] OF tyXMLTableDat;
	iXMLTableDataBrdAvlTtlIdx : INT;
	bConnected : BOOL;
	bHandshakeDone : BOOL;
	bOverWriteSlt : BOOL;
	bOverWriteWidth : BOOL;
	sReqRecipeNm : STRING[254];
	diReqWidthInUM : DINT;
	sInternalSnd : STRING[65535];
END_VAR
(**)
(*Local Input*)
VAR
	udiRstErr : UDINT := 0;
	bPrep : BOOL := TRUE;
	bEn : BOOL := TRUE;
	bDis : BOOL := FALSE;
	sIPAddr : STRING[15] := '192.168.0.100';
	uiClntPort : UINT := 0;
	tyDTStructure : DTStructure := (year:=2019,month:=01,day:=05,wday:=05,hour:=21,minute:=28,second:=30,millisec:=123,microsec:=456);
	dtCurrDT : DATE_AND_TIME := DT#2019-02-23-12:30:50;
	sVersion : STRING[7] := '5.00.0';
	sRecipeNm : STRING[254] := '';
	diWidthInUM : DINT := 0;
	udiSndBffrSize : UDINT := 65536;
	udiRcvBffrSize : UDINT := 65536;
	udiAliveIdleTimeInSec : UDINT := 5;
	tConnTimeOut : TIME := T#30s;
	diTransferInTO : DINT := 30000;
	bOpsRun : BOOL := FALSE;
	bInterruptSen : BOOL := FALSE;
	udiFileKeepDay : UDINT := 30;
	sProgNm : STRING[15] := 'OpCon';
	bNtSettingsLoadDone : BOOL := TRUE;
	sInfoMsg : STRING[200];
	bInternalUse : BOOL;
	sInternalRcv : STRING[65535];
	a_tyProdRcpList : ARRAY[1..c_udiProdRcpMax] OF tyProdRcpParam;
	tyProdRcpCurrRcp : tyProdRcpParam;
END_VAR
(**)
(*Local*)
VAR
	bTestEn : BOOL;
	sSnd_0 : STRING[65535];
	fbFileFullWrite_0 : fbFileFullWrite;
	bRstErr : BOOL;
	udiRstErrOld : UDINT;
	bInitDone : BOOL;
	bInitialDone : BOOL;
	bRun : BOOL;
	bStop : BOOL;
	bRstConnection : BOOL;
	bRstState : BOOL;
	udiTCPIdent : UDINT;
	udiXMLTableWriteIdx : UDINT;
	udiMsgSendBffr : UDINT;
	udiSndMsgLen : UDINT;
	i : INT;
	bMsgIssued : ARRAY[1..15] OF BOOL;
	sSnd : STRING[65535];
	sRcv : STRING[65535];
	a_tyXMLTableDataRcv : ARRAY[0..200] OF tyXMLTableDat;
	a_tyXMLTableDataSnd : ARRAY[0..200] OF tyXMLTableDat;
	a_eMsgSend : ARRAY[0..50] OF eOpConMsgType;
	fbClntConnect : fbTCPClntConnect;
	fbRcv : fbTCPRcv;
	fbSend : fbTCPSnd;
	fbClose : fbTCPClose;
	fbParseXMLTable : fbOpConParseXMLTable;
	udiLogCntr : UDINT := 1;
	udiWriteLogCntr : UDINT := 1;
	a_sLogList : ARRAY[1..10] OF STRING[65535];
	sDT : STRING[80];
	dtCurrDTTemp : DATE_AND_TIME;
	fbFileAppend1 : fbFileFullAppend;
	fbFileOldDel1 : fbFileOldDel;
	s1 : {REDUND_UNREPLICABLE} ARRAY[1..15] OF STRING[80];
	sPLCErrorText : STRING[80];
	uiPLCErrorNo : UINT;
END_VAR
(*xml*)
VAR
	tyOpConEvent : tyEventType := (tyData:=(sVersion:='2.2',siEventSwitch:=-1,usiContentType:=3));
	tyOpConLocation : tyLocationParam;
	tyPartReceive : tyOpConPartReceive := (tyData:=(sTypeNo:='1111111111',sTypeVar:='0000',asDataType:='8'));
	tyPlcGrab : tyOpConPlcGrabReceive;
	tyPartProcessed : tyOpConPartProcessed := (tyData:=(usiResult:=1,sTypeVar:='0000',usiWorkingCode:=1,usiNioBits:=1,uiBatch:=1,sMachineID:='1',sName:=['Prog1.Name','Pitch','Magazine.Type','Magazine.Position','Magazine.Layer'],sDataType:=[3('8'),2('3')])); (*datatype 8: string, 3:int*)
	tyPLCError : tyOpConPLCError := (tyData:=(sTypeVar:='0000',usiErrorType:=1,usiErrorState:=1,usiOperationMode:=1,bModeOn:=TRUE,iChainNo:=999));
	tyPartMissing : tyOpConPartMissing := (tyData:=(usiMissingPart:=1,sTypeVar:='0000'));
	tyPLCJam : tyOpConPLCJam := (tyData:=(sTypeVar:='0000'));
	tyPLCGrab : tyOpConPLCGrab := (tyData:=(sMagazineNm:=['','Magazine1','Magazine2','Magazine3',''],sDataType:=['',3('8'),'']));
	eOpConMsgReq : eOpConMsgType;
END_VAR
```

### AutoRcp.typ - Do Not Change!!!
```iecst
(*2019-04-25*)
(*Action*)
(*input WorkOrder/Board available/boardforecast  to output ProdRcp*)
(*change Rcp for individual Magazine *)

TYPE
	tyWorkOrderParam : 	STRUCT
		sRcpNm : STRING[254];
		diWidthInUM : DINT;
		diWidthInUM2 : DINT;
		diIntvlCntr : DINT;
		diMinSltValue : DINT;
		diMaxSltValue : DINT;
		diPitch : DINT;
		diBrdPerSlt : DINT;
		usiMcMod : USINT;
		bTopToBtm : BOOL;
		bGapBwtnBrd : BOOL;
		bLongBrd : BOOL;
		diMinReqFreeBffr : DINT;
		sDisplayInfo : STRING[30];
		dtLastModified : DATE_AND_TIME;
		diMtrPshrExtSpd : DINT;
		diMtrPshrExtTorq : DINT;
		diPshrOffset : DINT;
	END_STRUCT;
END_TYPE

(*Loader , Input  -> Board Property*)
(*Unloader, Board Property -> Input*)

TYPE
	tyBoardProperty : 	STRUCT
		sWorkOrderId : STRING[80]; (*The work order for the production of PCB.*)
		sBatchId : STRING[80]; (*The batch id of a splitted work order.*)
		sBoardId : STRING[36]; (*Indicating the ID of the available board*)
		sBoardIdCreatedBy : STRING[80]; (*MachineId of the machine which created the BoardId (the first machine in a consecutive row of machines implementing this protocol). The MachineId is part of the Hermes Configuration.*)
		eFailedBoard : eHermesFailedBoard; (*A value of Unknown Board, Good Board & Failed Board*)
		sProductTypeId : STRING[254]; (*Identifies a collection of PCBs sharing common properties.*)
		eFlippedBoard : eHermesFlippedBoard; (*A value of Unknown Side, Top Side Up & Bottom Side Up.*)
		sTopBarcode : STRING[254]; (*The barcode of the top side of the PCB*)
		sBottomBarcode : STRING[254]; (*The barcode of the bottom side of the PCB*)
		rLength : REAL; (*The length of the PCB in millimeter.*)
		rWidth : REAL; (*The width of the PCB in millimeter.*)
		rThickness : REAL; (*The thickness of the PCB in millimeter.*)
		rConveyorSpeed : REAL; (*The conveyor speed preferred by the upstream machine in millimeter per second.*)
		rTopClearanceHeight : REAL; (*The clearance height for the top side of the PCB in millimeter.*)
		rBottomClearanceHeight : REAL; (*The clearance height for the bottom side of the PCB in millimeter.*)
		rWeight : REAL; (*The weight of the PCB in grams.*)
	END_STRUCT;
	tyMagProperties : 	STRUCT
		sRcpNm : STRING[254]; (*//Only used for We Fab*)
		diWidth : DINT;
		diPitch : DINT;
		diMinSlt : DINT;
		diMaxSlt : DINT;
		sTrailingBarcode : STRING[254]; (*0259E01, use trailing 10 character to compare Magazine*)
	END_STRUCT;
END_TYPE

(**)

TYPE
	eAutoRcpAction :
		(
		AutoRcpActIdle,
		AutoRcpActCreateDir,
		AutoRcpActReadRetain2, (*for Traverser*)
		AutoRcpActWriteRetain2, (*for Traverser*)
		AutoRcpActReadRetain,
		AutoRcpActWriteRetain
		);
END_TYPE
```

### AutoRcp.var - Change By Project
```iecst
(*2019-06-27*)
(**)
(*Action & State & Status*)
VAR
	p_AutoRcpStat : UDINT;
	p_AutoRcpStatus : UDINT;
END_VAR
(**)
(*Alarm*)
VAR
	p_AutoRcpAlmData : UDINT;
	p_AutoRcpInfoData : UDINT;
	p_AutoRcpInfoData1 : UDINT;
END_VAR
(**)
(*Output*)
VAR
	p_AutoRcpUSAllow : UDINT;
	p_AutoRcpDSAllow : UDINT;
	p_AutoRcpProdAccDataMnl : UDINT;
	p_AutoRcpProdUpdtDataMnl : UDINT;
	p_AutoRcpMagAccDataMnl : UDINT;
	p_AutoRcpTimeAct : UDINT;
	p_AutoRcpSetDT : UDINT;
	p_AutoRcpWaitRlsBrd : UDINT;
	p_AutoRcpUpdtProdRcp : UDINT;
	p_AutoRcpProdRcpDiff : UDINT;
	p_AutoRcpCurrRcpProdID : UDINT;
	p_AutoRcpCurrRcpWidth : UDINT;
	p_AutoRcpbTravWidthDiffblk : UDINT;
	p_AutoRcpbMagChangeOverBlk : UDINT;
	p_AutoRcpbMag1PropDiffBlk : UDINT;
	p_AutoRcpbMag2PropDiffBlk : UDINT;
	p_AutoRcpbMag3PropDiffBlk : UDINT;
	p_AutoRcpbMag1WidthChg : UDINT;
	p_AutoRcpbMag2WidthChg : UDINT;
	p_AutoRcpbMag3WidthChg : UDINT;
	p_AutoRcpbMag1SlotChg : UDINT;
	p_AutoRcpbMag2SlotChg : UDINT;
	p_AutoRcpbMag3SlotChg : UDINT;
END_VAR
(*TravLif Width*)
VAR
	p_diAutoRcpTravLifWidth : UDINT;
END_VAR
(*Magazine Properties*)
VAR
	p_diAutoRcpAllMagProps : UDINT;
	p_diAutoRcpBrdProps : UDINT;
	p_diAutoRcpMag1MaxSlt : UDINT;
	p_diAutoRcpMag1MinSlt : UDINT;
	p_diAutoRcpMag1Pitch : UDINT;
	p_diAutoRcpMag1Width : UDINT;
	p_diAutoRcpMag2MaxSlt : UDINT;
	p_diAutoRcpMag2MinSlt : UDINT;
	p_diAutoRcpMag2Pitch : UDINT;
	p_diAutoRcpMag2Width : UDINT;
	p_diAutoRcpMag3MaxSlt : UDINT;
	p_diAutoRcpMag3MinSlt : UDINT;
	p_diAutoRcpMag3Pitch : UDINT;
	p_diAutoRcpMag3Width : UDINT;
	p_AutoRcpForceExitMag : UDINT;
END_VAR
```

### Program Logical/AutoRcp/AutoRcp (IEC, version 1.00.0) - place into CPUsw

#### Package Logical/AutoRcp/AutoRcp/PrecededBySelf - Intended for F1,F2

#### PrecededBySelfInitial.st
```iecst
ACTION PrecededBySelfInitial:

	//Mag Detail (Hermes)
	fbFileRead1.sDevice			:= 'Retain';
	fbFileRead1.sFile			:= 'MagazineRcp';
	fbFileRead1.udiOffset		:= 0;
	fbFileRead1.p_Dest			:= ADR(a_tyCurrZ2Rcp);
	fbFileRead1.udiLen			:= SIZEOF(a_tyCurrZ2Rcp);
	fbFileRead1(bEn := FALSE);

	fbFileWrite1.sDevice	:= 'Retain';
	fbFileWrite1.sFile			:= 'MagazineRcp';
	fbFileWrite1.udiOffset		:= 0;
	fbFileWrite1.p_Src			:= ADR(a_tyZ2RcpWr);
	fbFileWrite1.udiLen			:= SIZEOF(a_tyZ2RcpWr);
	fbFileWrite1.udiOption		:= 0;
	fbFileWrite1(bEn := FALSE);

	//Trav Detail (Hermes)
	fbFileRead2.sDevice			:= 'Retain';
	fbFileRead2.sFile			:= 'TravRcp';
	fbFileRead2.udiOffset		:= 0;
	fbFileRead2.p_Dest			:= ADR(tyCurrZ1Rcp);
	fbFileRead2.udiLen			:= SIZEOF(tyCurrZ1Rcp);
	fbFileRead2(bEn := FALSE);

	fbFileWrite2.sDevice	:= 'Retain';
	fbFileWrite2.sFile			:= 'TravRcp';
	fbFileWrite2.udiOffset		:= 0;
	fbFileWrite2.p_Src			:= ADR(tyZ1RcpWr);
	fbFileWrite2.udiLen			:= SIZEOF(tyZ1RcpWr);
	fbFileWrite2.udiOption		:= 0;
	fbFileWrite2(bEn := FALSE);

END_ACTION
```

#### PrecededBySelfLink.st
```iecst
ACTION PrecededBySelfLink:

	//For Accepting BA or BF from HermesA/B
	p_bHermesBADataAccepted := p_bHermesABAAccepted OR p_bHermesBBAAccepted;
	IF p_bHermesABAAccepted THEN
		p_tyHermesBARcv ACCESS p_USHermesABoardAvailableRcv;
	ELSIF  p_bHermesBBAAccepted THEN
		p_tyHermesBARcv ACCESS p_USHermesABoardAvailableRcv;
	END_IF

	p_bHermesBFDataAccepted	:= 	p_bHermesABFAccepted OR p_bHermesBBFAccepted;
	IF p_bHermesABFAccepted THEN
		p_tyHermesBFRcv ACCESS p_USHermesABoardForecastRcv;
	ELSIF p_bHermesBBFAccepted THEN
		p_tyHermesBFRcv ACCESS p_USHermesBBoardForecastRcv;
	END_IF

	//Z1 Accepting Condition
	p_bZ1AccNewRcpCondition := (p_bLinkOpsRun = TRUE) AND (p_bLinkOpsTravLifULInitDone = TRUE) AND (p_bLinkPshrConvHvBrd = FALSE);

	//Z2 Accepting Condition
	p_bZ2AccNewRcpCondition := (p_bLinkOpsRun = TRUE);// AND (p_bLinkOpsMagConvUL1InitDone AND p_bLinkOpsMagConvUL2InitDone AND p_bLinkOpsMagConvUL3InitDone);

END_ACTION
```
